C07276=1075.846,98.114,431.514,173.695,23.921,154.199
C07277=1075.840,97.865,431.531,173.693,23.918,154.199
C07278=1075.835,97.616,431.551,173.692,23.916,154.199
C07279=1075.829,97.367,431.568,173.691,23.913,154.198
C07280=1075.823,97.118,431.587,173.688,23.910,154.198
C07281=1075.817,96.868,431.605,173.687,23.908,154.198
C07282=1075.812,96.619,431.624,173.686,23.906,154.198
C07283=1075.805,96.370,431.642,173.683,23.903,154.197
C07284=1075.800,96.121,431.660,173.682,23.901,154.197
C07285=1075.794,95.871,431.678,173.681,23.898,154.197
C07286=1075.789,95.622,431.697,173.679,23.896,154.196
C07287=1075.782,95.341,431.718,173.677,23.893,154.196
C07288=1075.775,95.059,431.738,173.675,23.890,154.196
C07289=1075.770,94.778,431.759,173.674,23.887,154.196
C07290=1075.763,94.497,431.780,173.672,23.884,154.195
C07291=1075.757,94.248,431.797,173.670,23.882,154.195
C07292=1075.751,93.998,431.815,173.669,23.879,154.195
C07293=1075.746,93.749,431.835,173.667,23.877,154.194
C07294=1075.740,93.500,431.852,173.665,23.874,154.194
C07295=1075.734,93.250,431.870,173.664,23.872,154.194
C07296=1075.729,93.001,431.889,173.662,23.869,154.193
C07297=1075.723,92.752,431.907,173.661,23.866,154.193
C07298=1075.717,92.503,431.924,173.659,23.864,154.193
C07299=1075.711,92.253,431.944,173.657,23.861,154.192
C07300=1075.706,92.004,431.961,173.656,23.859,154.192
C07301=1075.700,91.754,431.979,173.655,23.856,154.192
C07302=1075.695,91.506,431.998,173.653,23.854,154.192
C07303=1075.689,91.257,432.016,173.651,23.851,154.191
C07304=1075.683,91.007,432.034,173.650,23.848,154.191
C07305=1075.677,90.758,432.052,173.648,23.846,154.191
C07306=1075.672,90.508,432.070,173.646,23.843,154.190
C07307=1075.666,90.259,432.088,173.645,23.841,154.190
C07308=1075.660,90.010,432.106,173.644,23.838,154.190
C07309=1075.654,89.760,432.124,173.642,23.836,154.190
C07310=1075.648,89.511,432.142,173.640,23.833,154.189
C07311=1075.642,89.262,432.160,173.639,23.831,154.189
C07312=1075.637,89.013,432.178,173.637,23.829,154.189
C07313=1075.630,88.764,432.196,173.635,23.826,154.188
C07314=1075.625,88.514,432.214,173.634,23.823,154.188
C07315=1075.619,88.264,432.232,173.632,23.821,154.188
C07316=1075.614,88.015,432.250,173.630,23.818,154.188
C07317=1075.608,87.766,432.267,173.629,23.816,154.187
C07318=1075.602,87.517,432.285,173.628,23.814,154.187
C07319=1075.596,87.268,432.304,173.626,23.811,154.187
C07320=1075.590,87.018,432.322,173.624,23.808,154.186
C07321=1075.585,86.769,432.339,173.623,23.806,154.186
C07322=1075.579,86.520,432.357,173.622,23.803,154.186
C07323=1075.573,86.271,432.375,173.620,23.801,154.185
C07324=1075.567,86.021,432.393,173.618,23.798,154.185
C07325=1075.561,85.772,432.410,173.617,23.796,154.185
C07326=1075.555,85.523,432.429,173.615,23.793,154.185
C07327=1075.549,85.274,432.446,173.613,23.791,154.184
C07328=1075.544,85.025,432.464,173.612,23.788,154.184
C07329=1075.538,84.775,432.482,173.611,23.785,154.184
C07330=1075.532,84.526,432.499,173.609,23.783,154.183
C07331=1075.527,84.276,432.518,173.607,23.780,154.183
C07332=1075.521,84.027,432.536,173.606,23.778,154.183
C07333=1075.516,83.778,432.553,173.604,23.775,154.183
C07334=1075.510,83.528,432.571,173.603,23.773,154.182
C07335=1075.504,83.279,432.589,173.601,23.770,154.182
C07336=1075.498,83.029,432.607,173.600,23.767,154.182
C07337=1075.493,82.780,432.624,173.598,23.765,154.181
C07338=1075.487,82.531,432.642,173.596,23.762,154.181
C07339=1075.481,82.281,432.660,173.595,23.760,154.181
C07340=1075.475,82.032,432.677,173.593,23.757,154.180
C07341=1075.470,81.783,432.695,173.592,23.755,154.180
C07342=1075.464,81.534,432.713,173.590,23.752,154.180
C07343=1075.458,81.285,432.730,173.589,23.749,154.180
C07344=1075.453,81.035,432.748,173.587,23.747,154.179
C07345=1075.447,80.786,432.766,173.586,23.745,154.179
C07346=1075.441,80.537,432.783,173.584,23.742,154.179
C07347=1075.436,80.288,432.801,173.583,23.739,154.178
C07348=1075.430,80.038,432.819,173.581,23.736,154.178
C07349=1075.424,79.789,432.836,173.580,23.734,154.178
C07350=1075.419,79.539,432.853,173.578,23.731,154.177
C07351=1075.412,79.258,432.874,173.577,23.728,154.177
C07352=1075.405,78.977,432.893,173.574,23.726,154.177
C07353=1075.399,78.696,432.912,173.573,23.723,154.176
C07354=1075.392,78.414,432.933,173.571,23.720,154.176
C07355=1075.387,78.165,432.950,173.570,23.718,154.176
C07356=1075.381,77.916,432.968,173.569,23.715,154.175
C07357=1075.375,77.666,432.986,173.566,23.712,154.175
C07358=1075.369,77.417,433.002,173.565,23.710,154.175
C07359=1075.364,77.168,433.020,173.564,23.707,154.175
C07360=1075.358,76.918,433.038,173.562,23.705,154.174
C07361=1075.352,76.669,433.055,173.560,23.702,154.174
C07362=1075.346,76.420,433.073,173.559,23.700,154.174
C07363=1075.340,76.170,433.089,173.558,23.697,154.173
C07364=1075.334,75.921,433.107,173.556,23.694,154.173
C07365=1075.329,75.672,433.124,173.554,23.692,154.173
C07366=1075.323,75.422,433.142,173.553,23.689,154.172
C07367=1075.317,75.173,433.159,173.552,23.687,154.172
C07368=1075.311,74.924,433.176,173.550,23.684,154.172
C07369=1075.306,74.675,433.194,173.548,23.682,154.172
C07370=1075.300,74.425,433.212,173.547,23.679,154.171
C07371=1075.294,74.176,433.228,173.546,23.676,154.171
C07372=1075.288,73.926,433.246,173.544,23.674,154.171
C07373=1075.282,73.677,433.263,173.542,23.671,154.170
C07374=1075.277,73.427,433.280,173.541,23.669,154.170
C07375=1075.271,73.178,433.297,173.539,23.666,154.170
C07376=1075.265,72.929,433.315,173.538,23.664,154.170
C07377=1075.259,72.680,433.333,173.536,23.661,154.169
C07378=1075.254,72.430,433.350,173.535,23.658,154.169
C07379=1075.247,72.181,433.367,173.533,23.656,154.169
C07380=1075.242,71.932,433.383,173.532,23.653,154.168
C07381=1075.236,71.682,433.401,173.531,23.651,154.168
C07382=1075.230,71.433,433.418,173.529,23.648,154.168
C07383=1075.225,71.183,433.435,173.527,23.645,154.167
C07384=1075.219,70.934,433.453,173.526,23.643,154.167
C07385=1075.214,70.685,433.470,173.525,23.641,154.167
C07386=1075.207,70.435,433.487,173.523,23.638,154.166
C07387=1075.202,70.186,433.505,173.521,23.635,154.166
C07388=1075.196,69.937,433.521,173.520,23.633,154.166
C07389=1075.190,69.688,433.538,173.519,23.630,154.165
C07390=1075.184,69.437,433.556,173.517,23.627,154.165
C07391=1075.178,69.189,433.573,173.515,23.625,154.165
C07392=1075.173,68.940,433.590,173.514,23.623,154.165
C07393=1075.167,68.690,433.607,173.513,23.620,154.164
C07394=1075.161,68.441,433.624,173.511,23.617,154.164
C07395=1075.155,68.191,433.641,173.509,23.615,154.164
C07396=1075.149,67.942,433.658,173.508,23.612,154.163
C07397=1075.144,67.693,433.675,173.507,23.610,154.163
C07398=1075.138,67.444,433.693,173.505,23.607,154.163
C07399=1075.132,67.194,433.709,173.503,23.605,154.163
C07400=1075.126,66.944,433.727,173.502,23.602,154.162
C07401=1075.120,66.695,433.743,173.501,23.599,154.162
C07402=1075.115,66.446,433.761,173.499,23.597,154.162
C07403=1075.109,66.197,433.777,173.497,23.594,154.161
C07404=1075.104,65.947,433.794,173.496,23.592,154.161
C07405=1075.097,65.698,433.811,173.495,23.589,154.161
C07406=1075.091,65.448,433.828,173.493,23.586,154.160
C07407=1075.085,65.199,433.845,173.492,23.584,154.160
C07408=1075.080,64.950,433.862,173.490,23.581,154.160
C07409=1075.074,64.701,433.879,173.489,23.579,154.160
C07410=1075.069,64.451,433.896,173.487,23.576,154.159
C07411=1075.063,64.202,433.912,173.486,23.573,154.159
C07412=1075.056,63.952,433.930,173.485,23.571,154.159
C07413=1075.050,63.703,433.946,173.483,23.568,154.158
C07414=1075.044,63.454,433.963,173.481,23.566,154.158
C07415=1075.038,63.173,433.982,173.480,23.564,154.158
C07416=1075.031,62.892,434.000,173.478,23.560,154.157
C07417=1075.024,62.609,434.020,173.477,23.558,154.157
C07418=1075.018,62.328,434.039,173.475,23.555,154.157
C07419=1075.012,62.079,434.055,173.473,23.552,154.156
C07420=1075.006,61.830,434.071,173.472,23.550,154.156
C07421=1075.000,61.580,434.089,173.470,23.547,154.156
C07422=1074.994,61.330,434.106,173.468,23.545,154.156
C07423=1074.988,61.081,434.122,173.467,23.542,154.155
C07424=1074.983,60.831,434.139,173.466,23.540,154.155
C07425=1074.976,60.583,434.156,173.465,23.537,154.155
C07426=1074.970,60.333,434.172,173.462,23.534,154.154
C07427=1074.964,60.084,434.188,173.461,23.532,154.154
C07428=1074.959,59.834,434.205,173.460,23.529,154.154
C07429=1074.952,59.585,434.222,173.459,23.527,154.153
C07430=1074.946,59.336,434.239,173.457,23.524,154.153
C07431=1074.941,59.086,434.255,173.455,23.522,154.153
C07432=1074.935,58.837,434.272,173.454,23.519,154.153
C07433=1074.929,58.588,434.289,173.453,23.516,154.152
C07434=1074.923,58.338,434.305,173.451,23.514,154.152
C07435=1074.918,58.089,434.322,173.450,23.512,154.152
C07436=1074.912,57.839,434.338,173.448,23.509,154.151
C07437=1074.906,57.590,434.354,173.446,23.506,154.151
C07438=1074.900,57.341,434.371,173.445,23.504,154.151
C07439=1074.894,57.091,434.388,173.444,23.502,154.150
C07440=1074.888,56.842,434.405,173.443,23.499,154.150
C07441=1074.882,56.592,434.421,173.440,23.496,154.150
C07442=1074.876,56.343,434.437,173.439,23.493,154.150
C07443=1074.871,56.093,434.454,173.438,23.491,154.149
C07444=1074.865,55.844,434.470,173.437,23.489,154.149
C07445=1074.859,55.595,434.487,173.435,23.486,154.149
C07446=1074.853,55.345,434.503,173.433,23.483,154.148
C07447=1074.847,55.097,434.520,173.432,23.481,154.148
C07448=1074.841,54.847,434.537,173.431,23.478,154.148
C07449=1074.836,54.598,434.553,173.429,23.476,154.147
C07450=1074.830,54.348,434.569,173.428,23.473,154.147
C07451=1074.824,54.099,434.585,173.426,23.470,154.147
C07452=1074.818,53.849,434.602,173.425,23.468,154.146
C07453=1074.812,53.600,434.619,173.423,23.465,154.146
C07454=1074.807,53.350,434.635,173.422,23.463,154.146
C07455=1074.801,53.101,434.651,173.421,23.460,154.146
C07456=1074.795,52.852,434.667,173.419,23.457,154.145
C07457=1074.789,52.602,434.684,173.417,23.455,154.145
C07458=1074.783,52.353,434.700,173.416,23.452,154.145
C07459=1074.777,52.103,434.717,173.415,23.450,154.144
C07460=1074.772,51.854,434.733,173.414,23.447,154.144
C07461=1074.766,51.605,434.749,173.412,23.444,154.144
C07462=1074.760,51.355,434.765,173.410,23.442,154.143
C07463=1074.754,51.106,434.782,173.409,23.439,154.143
C07464=1074.748,50.856,434.799,173.408,23.437,154.143
C07465=1074.743,50.607,434.815,173.406,23.434,154.142
C07466=1074.737,50.358,434.831,173.404,23.431,154.142
C07467=1074.731,50.108,434.847,173.403,23.429,154.142
C07468=1074.725,49.859,434.864,173.402,23.426,154.142
C07469=1074.719,49.609,434.880,173.400,23.424,154.141
C07470=1074.714,49.360,434.897,173.399,23.421,154.141
C07471=1074.708,49.111,434.912,173.398,23.419,154.141
C07472=1074.703,48.861,434.928,173.396,23.416,154.140
C07473=1074.697,48.612,434.944,173.394,23.413,154.140
C07474=1074.691,48.363,434.961,173.393,23.411,154.140
C07475=1074.685,48.113,434.977,173.392,23.408,154.139
C07476=1074.679,47.864,434.994,173.391,23.406,154.139
C07477=1074.673,47.614,435.010,173.389,23.403,154.139
C07478=1074.668,47.365,435.026,173.387,23.400,154.138
C07479=1074.661,47.083,435.044,173.386,23.398,154.138
C07480=1074.655,46.801,435.062,173.384,23.394,154.138
C07481=1074.648,46.520,435.081,173.383,23.391,154.137
C07482=1074.642,46.238,435.099,173.381,23.389,154.137
C07483=1074.636,45.989,435.115,173.380,23.386,154.137
C07484=1074.630,45.739,435.131,173.378,23.383,154.136
C07485=1074.625,45.490,435.147,173.377,23.381,154.136
C07486=1074.619,45.241,435.163,173.376,23.378,154.136
C07487=1074.614,44.991,435.180,173.374,23.375,154.135
C07488=1074.608,44.742,435.196,173.372,23.373,154.135
C07489=1074.602,44.492,435.212,173.371,23.370,154.135
C07490=1074.596,44.243,435.228,173.370,23.367,154.134
C07491=1074.591,43.994,435.244,173.369,23.365,154.134
C07492=1074.585,43.744,435.259,173.367,23.362,154.134
C07493=1074.579,43.495,435.276,173.365,23.360,154.134
C07494=1074.573,43.245,435.292,173.364,23.357,154.133
C07495=1074.567,42.996,435.308,173.363,23.354,154.133
C07496=1074.562,42.746,435.324,173.362,23.352,154.133
C07497=1074.556,42.497,435.340,173.360,23.349,154.132
C07498=1074.549,42.248,435.356,173.359,23.347,154.132
C07499=1074.544,41.998,435.371,173.357,23.344,154.132
C07500=1074.538,41.749,435.387,173.356,23.341,154.131
C07501=1074.532,41.500,435.403,173.354,23.339,154.131
C07502=1074.526,41.250,435.419,173.353,23.337,154.131
C07503=1074.520,41.000,435.435,173.352,23.334,154.131
C07504=1074.515,40.751,435.451,173.350,23.332,154.130
C07505=1074.509,40.501,435.467,173.348,23.328,154.130
C07506=1074.504,40.252,435.483,173.347,23.326,154.130
C07507=1074.497,40.003,435.498,173.346,23.324,154.129
C07508=1074.491,39.753,435.514,173.345,23.321,154.129
C07509=1074.485,39.504,435.530,173.343,23.318,154.129
C07510=1074.480,39.254,435.546,173.341,23.315,154.128
C07511=1074.474,39.005,435.562,173.340,23.313,154.128
C07512=1074.469,38.755,435.577,173.339,23.311,154.128
C07513=1074.463,38.506,435.593,173.337,23.308,154.127
C07514=1074.457,38.256,435.609,173.336,23.305,154.127
C07515=1074.450,38.007,435.625,173.335,23.303,154.127
C07516=1074.445,37.758,435.640,173.333,23.300,154.127
C07517=1074.439,37.508,435.656,173.332,23.298,154.126
C07518=1074.433,37.259,435.672,173.330,23.295,154.126
C07519=1074.427,37.009,435.687,173.329,23.293,154.126
C07520=1074.421,36.760,435.703,173.328,23.290,154.125
C07521=1074.415,36.510,435.719,173.327,23.287,154.125
C07522=1074.409,36.262,435.734,173.324,23.285,154.125
C07523=1074.404,36.012,435.750,173.323,23.282,154.124
C07524=1074.398,35.762,435.766,173.322,23.280,154.124
C07525=1074.392,35.513,435.782,173.320,23.277,154.124
C07526=1074.386,35.263,435.797,173.319,23.275,154.124
C07527=1074.380,35.014,435.812,173.318,23.272,154.123
C07528=1074.375,34.764,435.828,173.316,23.269,154.123
C07529=1074.368,34.515,435.844,173.315,23.267,154.123
C07530=1074.362,34.265,435.859,173.313,23.264,154.122
C07531=1074.357,34.017,435.875,173.312,23.262,154.122
C07532=1074.351,33.767,435.890,173.311,23.260,154.122
C07533=1074.345,33.517,435.906,173.309,23.257,154.121
C07534=1074.339,33.268,435.922,173.308,23.254,154.121
C07535=1074.333,33.019,435.936,173.306,23.251,154.121
C07536=1074.327,32.769,435.953,173.305,23.249,154.120
C07537=1074.322,32.519,435.968,173.304,23.247,154.120
C07538=1074.315,32.270,435.983,173.302,23.244,154.120
C07539=1074.310,32.021,435.999,173.301,23.242,154.120
C07540=1074.304,31.771,436.015,173.300,23.239,154.119
C07541=1074.298,31.521,436.030,173.298,23.236,154.119
C07542=1074.292,31.272,436.046,173.296,23.234,154.119
C07543=1074.285,30.991,436.063,173.295,23.231,154.118
C07544=1074.279,30.709,436.080,173.293,23.228,154.118
C07545=1074.272,30.427,436.098,173.292,23.225,154.118
C07546=1074.265,30.146,436.115,173.291,23.222,154.117
C07547=1074.260,29.897,436.130,173.289,23.220,154.117
C07548=1074.255,29.647,436.146,173.287,23.217,154.117
C07549=1074.248,29.398,436.161,173.286,23.214,154.116
C07550=1074.243,29.148,436.177,173.285,23.212,154.116
C07551=1074.237,28.898,436.192,173.284,23.209,154.116
C07552=1074.230,28.649,436.208,173.282,23.207,154.116
C07553=1074.225,28.400,436.223,173.280,23.204,154.115
C07554=1074.219,28.150,436.238,173.279,23.201,154.115
C07555=1074.213,27.900,436.253,173.278,23.199,154.115
C07556=1074.207,27.651,436.268,173.276,23.196,154.114
C07557=1074.202,27.402,436.284,173.275,23.194,154.114
C07558=1074.195,27.152,436.299,173.274,23.192,154.114
C07559=1074.190,26.902,436.315,173.273,23.189,154.113
C07560=1074.184,26.653,436.329,173.270,23.186,154.113
C07561=1074.178,26.404,436.345,173.269,23.184,154.113
C07562=1074.172,26.154,436.360,173.268,23.181,154.112
C07563=1074.166,25.906,436.375,173.267,23.178,154.112
C07564=1074.160,25.656,436.391,173.265,23.176,154.112
C07565=1074.154,25.406,436.406,173.264,23.174,154.112
C07566=1074.149,25.157,436.421,173.263,23.171,154.111
C07567=1074.142,24.907,436.436,173.261,23.168,154.111
C07568=1074.137,24.657,436.451,173.259,23.166,154.111
C07569=1074.131,24.409,436.467,173.258,23.164,154.111
C07570=1074.124,24.159,436.481,173.257,23.161,154.110
C07571=1074.119,23.909,436.497,173.256,23.158,154.110
C07572=1074.113,23.660,436.512,173.255,23.156,154.110
C07573=1074.107,23.410,436.527,173.252,23.153,154.109
C07574=1074.101,23.160,436.542,173.251,23.151,154.109
C07575=1074.095,22.912,436.557,173.250,23.148,154.109
C07576=1074.089,22.662,436.572,173.248,23.146,154.108
C07577=1074.083,22.413,436.587,173.247,23.143,154.108
C07578=1074.078,22.163,436.602,173.246,23.141,154.108
C07579=1074.071,21.913,436.617,173.245,23.138,154.107
C07580=1074.066,21.664,436.632,173.243,23.135,154.107
C07581=1074.060,21.414,436.647,173.241,23.133,154.107
C07582=1074.054,21.165,436.662,173.240,23.130,154.107
C07583=1074.049,20.915,436.678,173.239,23.128,154.106
C07584=1074.042,20.665,436.692,173.238,23.125,154.106
C07585=1074.036,20.417,436.707,173.236,23.123,154.106
C07586=1074.031,20.167,436.723,173.235,23.121,154.105
C07587=1074.025,19.918,436.737,173.233,23.118,154.105
C07588=1074.019,19.668,436.752,173.232,23.115,154.105
C07589=1074.013,19.418,436.768,173.230,23.112,154.105
C07590=1074.007,19.169,436.782,173.229,23.110,154.104
C07591=1074.001,18.919,436.797,173.228,23.108,154.104
C07592=1073.995,18.670,436.812,173.227,23.105,154.104
C07593=1073.989,18.420,436.827,173.225,23.103,154.103
C07594=1073.984,18.171,436.842,173.223,23.100,154.103
C07595=1073.977,17.922,436.857,173.222,23.097,154.103
C07596=1073.971,17.672,436.872,173.221,23.095,154.103
C07597=1073.966,17.423,436.887,173.219,23.093,154.102
C07598=1073.960,17.173,436.901,173.218,23.090,154.102
C07599=1073.954,16.924,436.916,173.217,23.088,154.102
C07600=1073.948,16.674,436.931,173.216,23.085,154.101
C07601=1073.943,16.425,436.946,173.214,23.082,154.101
C07602=1073.936,16.175,436.961,173.212,23.080,154.101
C07603=1073.930,15.926,436.975,173.211,23.077,154.100
C07604=1073.924,15.676,436.990,173.210,23.075,154.100
C07605=1073.919,15.427,437.006,173.208,23.072,154.100
C07606=1073.913,15.177,437.020,173.207,23.070,154.100
C07607=1073.906,14.897,437.036,173.205,23.066,154.099
C07608=1073.900,14.616,437.053,173.204,23.064,154.099
C07609=1073.893,14.337,437.069,173.203,23.062,154.099
C07610=1073.886,14.056,437.087,173.201,23.058,154.098
C07611=1073.881,13.807,437.101,173.199,23.056,154.098
C07612=1073.874,13.557,437.116,173.198,23.053,154.098
C07613=1073.868,13.308,437.130,173.197,23.051,154.097
C07614=1073.862,13.059,437.145,173.196,23.049,154.097
C07615=1073.856,12.808,437.159,173.194,23.046,154.097
C07616=1073.850,12.559,437.174,173.192,23.043,154.097
C07617=1073.844,12.310,437.189,173.191,23.041,154.096
C07618=1073.838,12.061,437.203,173.190,23.038,154.096
C07619=1073.832,11.810,437.218,173.188,23.036,154.096
C07620=1073.826,11.561,437.232,173.187,23.034,154.095
C07621=1073.820,11.312,437.247,173.186,23.031,154.095
C07622=1073.815,11.062,437.261,173.184,23.029,154.095
C07623=1073.808,10.813,437.276,173.182,23.026,154.095
C07624=1073.802,10.564,437.291,173.181,23.024,154.094
C07625=1073.796,10.313,437.305,173.180,23.021,154.094
C07626=1073.790,10.064,437.319,173.179,23.019,154.094
C07627=1073.784,9.815,437.334,173.177,23.016,154.094
C07628=1073.779,9.565,437.348,173.176,23.014,154.093
C07629=1073.772,9.316,437.363,173.175,23.011,154.093
C07630=1073.766,9.067,437.378,173.173,23.009,154.093
C07631=1073.760,8.816,437.392,173.171,23.006,154.092
C07632=1073.755,8.567,437.407,173.170,23.004,154.092
C07633=1073.748,8.318,437.421,173.169,23.002,154.092
C07634=1073.743,8.068,437.435,173.167,22.999,154.092
C07635=1073.736,7.818,437.450,173.166,22.997,154.091
C07636=1073.731,7.569,437.464,173.165,22.995,154.091
C07637=1073.725,7.320,437.479,173.163,22.992,154.091
C07638=1073.719,7.070,437.494,173.161,22.989,154.091
C07639=1073.713,6.821,437.508,173.160,22.987,154.090
C07640=1073.707,6.571,437.522,173.159,22.984,154.090
C07641=1073.701,6.321,437.536,173.158,22.982,154.090
C07642=1073.695,6.072,437.551,173.156,22.980,154.089
C07643=1073.690,5.822,437.565,173.155,22.977,154.089
C07644=1073.684,5.573,437.580,173.154,22.975,154.089
C07645=1073.678,5.323,437.594,173.152,22.972,154.089
C07646=1073.672,5.074,437.609,173.150,22.969,154.088
C07647=1073.666,4.824,437.623,173.149,22.967,154.088
C07648=1073.659,4.575,437.637,173.148,22.965,154.088
C07649=1073.654,4.326,437.651,173.146,22.962,154.087
C07650=1073.647,4.076,437.666,173.145,22.960,154.087
C07651=1073.642,3.826,437.679,173.144,22.957,154.087
C07652=1073.636,3.577,437.694,173.143,22.955,154.087
C07653=1073.630,3.327,437.708,173.141,22.952,154.086
C07654=1073.624,3.078,437.723,173.139,22.950,154.086
C07655=1073.618,2.828,437.737,173.138,22.947,154.086
C07656=1073.612,2.579,437.752,173.137,22.945,154.086
C07657=1073.607,2.329,437.765,173.135,22.942,154.085
C07658=1073.601,2.079,437.780,173.134,22.940,154.085
C07659=1073.595,1.830,437.794,173.133,22.937,154.085
C07660=1073.590,1.581,437.808,173.132,22.935,154.084
C07661=1073.583,1.331,437.823,173.130,22.933,154.084
C07662=1073.577,1.082,437.836,173.128,22.930,154.084
C07663=1073.572,0.832,437.850,173.127,22.927,154.084
C07664=1073.565,0.582,437.865,173.126,22.925,154.083
C07665=1073.560,0.333,437.879,173.124,22.922,154.083
C07666=1073.554,0.084,437.894,173.123,22.920,154.083
C07667=1073.548,-0.166,437.908,173.122,22.918,154.082
C07668=1073.542,-0.416,437.922,173.121,22.915,154.082
C07669=1073.537,-0.665,437.936,173.119,22.913,154.082
C07670=1073.531,-0.915,437.950,173.117,22.910,154.082
C07671=1073.524,-1.193,437.966,173.116,22.907,154.081
C07672=1073.517,-1.471,437.981,173.115,22.904,154.081
C07673=1073.511,-1.750,437.998,173.113,22.902,154.081
C07674=1073.504,-2.027,438.013,173.112,22.899,154.080
C07675=1073.498,-2.278,438.027,173.110,22.897,154.080
C07676=1073.493,-2.527,438.041,173.109,22.894,154.080
C07677=1073.487,-2.777,438.055,173.108,22.892,154.080
C07678=1073.482,-3.026,438.070,173.106,22.889,154.079
C07679=1073.476,-3.276,438.084,173.104,22.887,154.079
C07680=1073.469,-3.525,438.097,173.103,22.884,154.079
C07681=1073.464,-3.775,438.111,173.102,22.882,154.078
C07682=1073.457,-4.024,438.125,173.101,22.879,154.078
C07683=1073.451,-4.274,438.139,173.099,22.877,154.078
C07684=1073.446,-4.523,438.153,173.098,22.874,154.078
C07685=1073.439,-4.773,438.167,173.097,22.873,154.077
C07686=1073.433,-5.022,438.181,173.094,22.870,154.077
C07687=1073.428,-5.272,438.195,173.093,22.867,154.077
C07688=1073.422,-5.521,438.208,173.092,22.865,154.077
C07689=1073.415,-5.771,438.223,173.091,22.862,154.076
C07690=1073.409,-6.021,438.236,173.089,22.860,154.076
C07691=1073.404,-6.270,438.250,173.088,22.858,154.076
C07692=1073.397,-6.520,438.265,173.087,22.856,154.076
C07693=1073.391,-6.769,438.278,173.085,22.853,154.075
C07694=1073.386,-7.019,438.292,173.083,22.850,154.075
C07695=1073.379,-7.268,438.305,173.082,22.848,154.075
C07696=1073.373,-7.518,438.319,173.081,22.845,154.075
C07697=1073.368,-7.768,438.333,173.080,22.843,154.074
C07698=1073.362,-8.017,438.346,173.078,22.841,154.074
C07699=1073.356,-8.266,438.361,173.077,22.839,154.074
C07700=1073.349,-8.516,438.375,173.076,22.836,154.074
C07701=1073.344,-8.765,438.389,173.074,22.834,154.073
C07702=1073.338,-9.015,438.402,173.073,22.831,154.073
C07703=1073.332,-9.264,438.416,173.071,22.829,154.073
C07704=1073.326,-9.515,438.430,173.069,22.827,154.073
C07705=1073.320,-9.764,438.443,173.068,22.824,154.072
C07706=1073.314,-10.013,438.457,173.067,22.822,154.072
C07707=1073.308,-10.263,438.470,173.066,22.819,154.072
C07708=1073.302,-10.512,438.484,173.064,22.817,154.071
C07709=1073.296,-10.763,438.498,173.063,22.815,154.071
C07710=1073.290,-11.012,438.512,173.062,22.813,154.071
C07711=1073.285,-11.261,438.526,173.060,22.810,154.071
C07712=1073.278,-11.511,438.539,173.058,22.807,154.070
C07713=1073.273,-11.760,438.553,173.057,22.805,154.070
C07714=1073.266,-12.010,438.566,173.056,22.802,154.070
C07715=1073.261,-12.260,438.580,173.054,22.801,154.070
C07716=1073.254,-12.509,438.593,173.053,22.798,154.069
C07717=1073.249,-12.759,438.607,173.052,22.796,154.069
C07718=1073.243,-13.008,438.621,173.051,22.793,154.069
C07719=1073.237,-13.257,438.634,173.049,22.791,154.069
C07720=1073.231,-13.507,438.648,173.047,22.788,154.069
C07721=1073.225,-13.757,438.662,173.046,22.786,154.068
C07722=1073.220,-14.007,438.676,173.045,22.784,154.068
C07723=1073.213,-14.256,438.689,173.043,22.781,154.068
C07724=1073.208,-14.505,438.703,173.042,22.779,154.067
C07725=1073.202,-14.755,438.716,173.041,22.777,154.067
C07726=1073.196,-15.004,438.730,173.039,22.774,154.067
C07727=1073.190,-15.254,438.743,173.038,22.772,154.067
C07728=1073.183,-15.504,438.756,173.036,22.769,154.066
C07729=1073.178,-15.754,438.770,173.035,22.767,154.066
C07730=1073.172,-16.003,438.783,173.033,22.765,154.066
C07731=1073.166,-16.252,438.797,173.032,22.762,154.066
C07732=1073.160,-16.502,438.811,173.031,22.760,154.066
C07733=1073.154,-16.751,438.824,173.029,22.758,154.065
C07734=1073.147,-17.002,438.837,173.028,22.756,154.065
C07735=1073.141,-17.278,438.853,173.026,22.753,154.065
C07736=1073.135,-17.554,438.867,173.025,22.750,154.064
C07737=1073.127,-17.831,438.882,173.023,22.748,154.064
C07738=1073.121,-18.108,438.896,173.021,22.745,154.064
C07739=1073.115,-18.357,438.910,173.020,22.743,154.064
C07740=1073.109,-18.607,438.923,173.019,22.741,154.063
C07741=1073.103,-18.856,438.936,173.017,22.738,154.063
C07742=1073.098,-19.106,438.950,173.016,22.736,154.063
C07743=1073.091,-19.355,438.963,173.015,22.734,154.063
C07744=1073.085,-19.605,438.977,173.013,22.731,154.062
C07745=1073.079,-19.855,438.989,173.012,22.729,154.062
C07746=1073.073,-20.105,439.003,173.011,22.727,154.062
C07747=1073.067,-20.354,439.017,173.009,22.724,154.062
C07748=1073.061,-20.604,439.029,173.007,22.722,154.062
C07749=1073.056,-20.853,439.043,173.006,22.720,154.061
C07750=1073.049,-21.103,439.056,173.005,22.717,154.061
C07751=1073.043,-21.352,439.070,173.004,22.715,154.061
C07752=1073.037,-21.602,439.082,173.002,22.713,154.061
C07753=1073.032,-21.851,439.096,173.001,22.711,154.060
C07754=1073.026,-22.100,439.109,173.000,22.708,154.060
C07755=1073.020,-22.350,439.122,172.998,22.706,154.060
C07756=1073.013,-22.600,439.135,172.996,22.703,154.060
C07757=1073.008,-22.849,439.149,172.995,22.701,154.059
C07758=1073.001,-23.100,439.162,172.993,22.699,154.059
C07759=1072.995,-23.349,439.175,172.992,22.697,154.059
C07760=1072.990,-23.599,439.189,172.991,22.694,154.059
C07761=1072.984,-23.849,439.202,172.989,22.692,154.059
C07762=1072.978,-24.098,439.215,172.988,22.690,154.058
C07763=1072.971,-24.347,439.228,172.987,22.688,154.058
C07764=1072.966,-24.597,439.241,172.985,22.685,154.058
C07765=1072.960,-24.847,439.254,172.983,22.683,154.058
C07766=1072.954,-25.096,439.267,172.982,22.681,154.057
C07767=1072.948,-25.346,439.280,172.981,22.678,154.057
C07768=1072.942,-25.595,439.294,172.979,22.676,154.057
C07769=1072.937,-25.845,439.307,172.978,22.674,154.057
C07770=1072.930,-26.094,439.320,172.977,22.671,154.056
C07771=1072.924,-26.344,439.333,172.976,22.669,154.056
C07772=1072.918,-26.594,439.346,172.974,22.667,154.056
C07773=1072.913,-26.844,439.359,172.973,22.665,154.056
C07774=1072.907,-27.093,439.372,172.971,22.662,154.056
C07775=1072.901,-27.343,439.385,172.969,22.660,154.055
C07776=1072.895,-27.592,439.398,172.968,22.658,154.055
C07777=1072.889,-27.842,439.411,172.967,22.656,154.055
C07778=1072.883,-28.091,439.424,172.965,22.654,154.055
C07779=1072.877,-28.341,439.436,172.964,22.651,154.054
C07780=1072.870,-28.590,439.450,172.963,22.649,154.054
C07781=1072.865,-28.840,439.462,172.961,22.647,154.054
C07782=1072.858,-29.090,439.476,172.960,22.645,154.054
C07783=1072.852,-29.339,439.488,172.959,22.643,154.054
C07784=1072.846,-29.589,439.501,172.956,22.640,154.053
C07785=1072.840,-29.839,439.514,172.955,22.638,154.053
C07786=1072.834,-30.088,439.527,172.954,22.635,154.053
C07787=1072.828,-30.338,439.540,172.952,22.633,154.053
C07788=1072.822,-30.587,439.553,172.951,22.632,154.053
C07789=1072.816,-30.837,439.566,172.950,22.629,154.052
C07790=1072.810,-31.087,439.578,172.948,22.627,154.052
C07791=1072.804,-31.336,439.591,172.947,22.625,154.052
C07792=1072.799,-31.585,439.604,172.946,22.623,154.052
C07793=1072.792,-31.834,439.617,172.944,22.620,154.051
C07794=1072.787,-32.084,439.629,172.942,22.618,154.051
C07795=1072.781,-32.334,439.642,172.941,22.616,154.051
C07796=1072.774,-32.584,439.655,172.939,22.614,154.051
C07797=1072.768,-32.833,439.668,172.938,22.611,154.051
C07798=1072.762,-33.083,439.681,172.937,22.609,154.050
C07799=1072.756,-33.359,439.696,172.936,22.607,154.050
C07800=1072.749,-33.634,439.709,172.933,22.604,154.050
C07801=1072.743,-33.910,439.723,172.932,22.602,154.050
C07802=1072.736,-34.186,439.737,172.931,22.600,154.049
C07803=1072.730,-34.436,439.750,172.929,22.597,154.049
C07804=1072.724,-34.686,439.762,172.928,22.595,154.049
C07805=1072.717,-34.935,439.776,172.926,22.592,154.049
C07806=1072.712,-35.184,439.788,172.925,22.591,154.049
C07807=1072.706,-35.434,439.800,172.923,22.588,154.048
C07808=1072.700,-35.683,439.814,172.922,22.586,154.048
C07809=1072.694,-35.933,439.826,172.920,22.584,154.048
C07810=1072.688,-36.183,439.839,172.919,22.582,154.048
C07811=1072.682,-36.433,439.851,172.918,22.580,154.048
C07812=1072.676,-36.682,439.864,172.917,22.577,154.047
C07813=1072.670,-36.932,439.877,172.915,22.576,154.047
C07814=1072.665,-37.181,439.889,172.914,22.573,154.047
C07815=1072.659,-37.431,439.902,172.912,22.571,154.047
C07816=1072.653,-37.681,439.914,172.910,22.569,154.047
C07817=1072.647,-37.930,439.928,172.909,22.566,154.046
C07818=1072.640,-38.180,439.940,172.907,22.565,154.046
C07819=1072.634,-38.430,439.952,172.906,22.562,154.046
C07820=1072.629,-38.679,439.964,172.905,22.560,154.046
C07821=1072.623,-38.929,439.977,172.903,22.558,154.046
C07822=1072.617,-39.178,439.990,172.902,22.556,154.045
C07823=1072.610,-39.428,440.002,172.901,22.554,154.045
C07824=1072.604,-39.678,440.015,172.899,22.552,154.045
C07825=1072.598,-39.928,440.027,172.897,22.549,154.045
C07826=1072.593,-40.177,440.040,172.896,22.547,154.045
C07827=1072.586,-40.427,440.052,172.894,22.545,154.045
C07828=1072.580,-40.676,440.065,172.893,22.543,154.044
C07829=1072.574,-40.926,440.077,172.892,22.541,154.044
C07830=1072.568,-41.175,440.090,172.890,22.539,154.044
C07831=1072.562,-41.425,440.102,172.889,22.537,154.044
C07832=1072.556,-41.675,440.114,172.888,22.535,154.043
C07833=1072.550,-41.925,440.127,172.886,22.533,154.043
C07834=1072.545,-42.174,440.139,172.885,22.531,154.043
C07835=1072.538,-42.423,440.151,172.884,22.528,154.043
C07836=1072.532,-42.673,440.163,172.881,22.526,154.043
C07837=1072.526,-42.923,440.176,172.880,22.524,154.043
C07838=1072.520,-43.173,440.188,172.878,22.522,154.043
C07839=1072.514,-43.421,440.201,172.877,22.520,154.042
C07840=1072.508,-43.671,440.213,172.876,22.518,154.042
C07841=1072.502,-43.921,440.226,172.874,22.516,154.042
C07842=1072.495,-44.171,440.238,172.873,22.514,154.042
C07843=1072.490,-44.421,440.251,172.872,22.512,154.041
C07844=1072.484,-44.670,440.263,172.870,22.510,154.041
C07845=1072.478,-44.919,440.275,172.869,22.508,154.041
C07846=1072.472,-45.169,440.287,172.868,22.505,154.041
C07847=1072.466,-45.419,440.300,172.865,22.503,154.041
C07848=1072.459,-45.669,440.312,172.864,22.501,154.041
C07849=1072.454,-45.918,440.324,172.862,22.499,154.040
C07850=1072.448,-46.168,440.336,172.861,22.497,154.040
C07851=1072.441,-46.417,440.348,172.860,22.495,154.040
C07852=1072.435,-46.667,440.361,172.858,22.493,154.040
C07853=1072.430,-46.917,440.372,172.857,22.491,154.040
C07854=1072.424,-47.167,440.384,172.856,22.489,154.040
C07855=1072.418,-47.416,440.397,172.854,22.487,154.039
C07856=1072.413,-47.666,440.409,172.853,22.485,154.039
C07857=1072.406,-47.915,440.421,172.852,22.483,154.039
C07858=1072.400,-48.165,440.434,172.850,22.481,154.039
C07859=1072.394,-48.415,440.446,172.848,22.479,154.039
C07860=1072.388,-48.664,440.458,172.847,22.476,154.038
C07861=1072.382,-48.914,440.470,172.845,22.474,154.038
C07862=1072.376,-49.164,440.483,172.844,22.472,154.038
C07863=1072.370,-49.440,440.496,172.842,22.470,154.038
C07864=1072.363,-49.716,440.509,172.841,22.468,154.038
C07865=1072.357,-49.992,440.523,172.839,22.466,154.038
C07866=1072.350,-50.269,440.536,172.838,22.463,154.037
C07867=1072.344,-50.518,440.548,172.836,22.461,154.037
C07868=1072.338,-50.767,440.560,172.835,22.459,154.037
C07869=1072.331,-51.018,440.572,172.833,22.458,154.037
C07870=1072.325,-51.267,440.584,172.832,22.456,154.037
C07871=1072.319,-51.516,440.596,172.830,22.454,154.037
C07872=1072.313,-51.766,440.608,172.828,22.451,154.037
C07873=1072.307,-52.016,440.620,172.827,22.450,154.036
C07874=1072.300,-52.266,440.632,172.825,22.448,154.036
C07875=1072.294,-52.515,440.643,172.824,22.446,154.036
C07876=1072.289,-52.765,440.656,172.822,22.444,154.036
C07877=1072.282,-53.014,440.668,172.821,22.442,154.036
C07878=1072.275,-53.264,440.680,172.820,22.440,154.036
C07879=1072.270,-53.514,440.691,172.818,22.438,154.035
C07880=1072.264,-53.763,440.703,172.817,22.436,154.035
C07881=1072.258,-54.013,440.716,172.815,22.434,154.035
C07882=1072.252,-54.262,440.727,172.814,22.432,154.035
C07883=1072.245,-54.512,440.738,172.813,22.430,154.035
C07884=1072.239,-54.762,440.751,172.811,22.428,154.035
C07885=1072.233,-55.012,440.763,172.809,22.426,154.035
C07886=1072.227,-55.261,440.774,172.807,22.424,154.034
C07887=1072.221,-55.511,440.786,172.806,22.422,154.034
C07888=1072.214,-55.761,440.798,172.805,22.420,154.034
C07889=1072.209,-56.010,440.809,172.803,22.419,154.034
C07890=1072.203,-56.260,440.822,172.802,22.417,154.034
C07891=1072.196,-56.510,440.834,172.800,22.415,154.034
C07892=1072.190,-56.759,440.845,172.799,22.413,154.034
C07893=1072.184,-57.009,440.857,172.798,22.411,154.033
C07894=1072.178,-57.258,440.869,172.796,22.410,154.033
C07895=1072.172,-57.508,440.880,172.795,22.408,154.033
C07896=1072.165,-57.758,440.892,172.793,22.406,154.033
C07897=1072.160,-58.007,440.905,172.792,22.404,154.033
C07898=1072.154,-58.257,440.915,172.790,22.402,154.033
C07899=1072.147,-58.507,440.927,172.788,22.400,154.033
C07900=1072.142,-58.756,440.939,172.787,22.398,154.033
C07901=1072.136,-59.006,440.951,172.785,22.396,154.032
C07902=1072.129,-59.255,440.963,172.784,22.394,154.032
C07903=1072.123,-59.505,440.974,172.782,22.392,154.032
C07904=1072.117,-59.755,440.986,172.781,22.390,154.032
C07905=1072.111,-60.004,440.997,172.780,22.388,154.032
C07906=1072.105,-60.254,441.009,172.778,22.387,154.032
C07907=1072.099,-60.504,441.021,172.777,22.385,154.032
C07908=1072.093,-60.753,441.032,172.775,22.383,154.031
C07909=1072.087,-61.003,441.044,172.774,22.381,154.031
C07910=1072.081,-61.252,441.055,172.772,22.379,154.031
C07911=1072.075,-61.502,441.068,172.771,22.377,154.031
C07912=1072.069,-61.752,441.079,172.769,22.375,154.031
C07913=1072.062,-62.001,441.091,172.768,22.373,154.031
C07914=1072.056,-62.251,441.102,172.766,22.371,154.031
C07915=1072.051,-62.501,441.114,172.764,22.370,154.031
C07916=1072.045,-62.751,441.125,172.763,22.368,154.030
C07917=1072.038,-63.000,441.137,172.761,22.366,154.030
C07918=1072.032,-63.250,441.148,172.760,22.364,154.030
C07919=1072.027,-63.499,441.160,172.759,22.362,154.030
C07920=1072.020,-63.749,441.172,172.757,22.360,154.030
C07921=1072.014,-63.999,441.183,172.756,22.359,154.030
C07922=1072.008,-64.248,441.195,172.754,22.357,154.030
C07923=1072.002,-64.499,441.206,172.753,22.355,154.029
C07924=1071.996,-64.748,441.218,172.751,22.353,154.029
C07925=1071.990,-64.998,441.229,172.750,22.351,154.029
C07926=1071.984,-65.247,441.241,172.748,22.349,154.029
C07927=1071.978,-65.524,441.254,172.746,22.347,154.029
C07928=1071.971,-65.802,441.267,172.745,22.345,154.029
C07929=1071.964,-66.080,441.279,172.743,22.343,154.029
C07930=1071.957,-66.357,441.292,172.742,22.341,154.028
C07931=1071.952,-66.607,441.303,172.740,22.340,154.028
C07932=1071.946,-66.857,441.314,172.738,22.337,154.028
C07933=1071.940,-67.106,441.326,172.737,22.335,154.028
C07934=1071.933,-67.356,441.337,172.735,22.334,154.028
C07935=1071.928,-67.606,441.348,172.734,22.332,154.028
C07936=1071.922,-67.855,441.361,172.732,22.330,154.028
C07937=1071.916,-68.105,441.372,172.731,22.328,154.028
C07938=1071.910,-68.355,441.383,172.729,22.326,154.028
C07939=1071.904,-68.604,441.394,172.728,22.324,154.027
C07940=1071.897,-68.854,441.406,172.727,22.323,154.027
C07941=1071.892,-69.104,441.416,172.725,22.321,154.027
C07942=1071.886,-69.353,441.429,172.724,22.319,154.027
C07943=1071.880,-69.603,441.440,172.722,22.317,154.027
C07944=1071.874,-69.853,441.451,172.721,22.315,154.027
C07945=1071.868,-70.102,441.463,172.719,22.314,154.027
C07946=1071.862,-70.352,441.474,172.718,22.312,154.027
C07947=1071.856,-70.602,441.485,172.716,22.310,154.027
C07948=1071.851,-70.852,441.496,172.715,22.309,154.026
C07949=1071.844,-71.100,441.508,172.713,22.307,154.026
C07950=1071.838,-71.351,441.519,172.712,22.305,154.026
C07951=1071.832,-71.600,441.530,172.711,22.303,154.026
C07952=1071.826,-71.850,441.541,172.708,22.301,154.026
C07953=1071.820,-72.100,441.552,172.707,22.299,154.026
C07954=1071.815,-72.349,441.564,172.705,22.298,154.026
C07955=1071.809,-72.599,441.576,172.704,22.296,154.026
C07956=1071.803,-72.849,441.587,172.702,22.294,154.026
C07957=1071.797,-73.098,441.597,172.701,22.292,154.025
C07958=1071.791,-73.348,441.609,172.699,22.290,154.025
C07959=1071.785,-73.597,441.620,172.698,22.289,154.025
C07960=1071.778,-73.847,441.631,172.696,22.287,154.025
C07961=1071.773,-74.097,441.642,172.695,22.285,154.025
C07962=1071.767,-74.346,441.653,172.693,22.284,154.025
C07963=1071.761,-74.597,441.664,172.692,22.282,154.025
C07964=1071.755,-74.846,441.675,172.690,22.281,154.025
C07965=1071.749,-75.096,441.687,172.689,22.279,154.025
C07966=1071.743,-75.345,441.698,172.687,22.277,154.025
C07967=1071.737,-75.595,441.709,172.686,22.275,154.024
C07968=1071.730,-75.845,441.720,172.684,22.274,154.024
C07969=1071.725,-76.094,441.731,172.683,22.272,154.024
C07970=1071.718,-76.345,441.742,172.681,22.271,154.024
C07971=1071.713,-76.594,441.753,172.680,22.269,154.024
C07972=1071.707,-76.844,441.764,172.678,22.267,154.024
C07973=1071.700,-77.093,441.775,172.677,22.265,154.024
C07974=1071.694,-77.343,441.786,172.675,22.264,154.024
C07975=1071.688,-77.592,441.797,172.674,22.262,154.024
C07976=1071.682,-77.843,441.808,172.672,22.260,154.024
C07977=1071.676,-78.092,441.819,172.670,22.259,154.024
C07978=1071.670,-78.342,441.830,172.669,22.257,154.024
C07979=1071.664,-78.592,441.841,172.667,22.255,154.024
C07980=1071.658,-78.841,441.852,172.666,22.254,154.024
C07981=1071.652,-79.091,441.864,172.664,22.252,154.023
C07982=1071.646,-79.340,441.875,172.663,22.251,154.023
C07983=1071.640,-79.589,441.885,172.661,22.249,154.023
C07984=1071.633,-79.840,441.896,172.660,22.247,154.023
C07985=1071.627,-80.089,441.907,172.658,22.245,154.023
C07986=1071.622,-80.339,441.917,172.657,22.244,154.023
C07987=1071.615,-80.589,441.928,172.655,22.243,154.023
C07988=1071.609,-80.839,441.939,172.654,22.241,154.023
C07989=1071.603,-81.088,441.949,172.652,22.239,154.023
C07990=1071.597,-81.338,441.961,172.650,22.238,154.023
C07991=1071.590,-81.617,441.973,172.649,22.236,154.023
C07992=1071.583,-81.897,441.985,172.647,22.235,154.023
C07993=1071.576,-82.177,441.997,172.645,22.232,154.023
C07994=1071.569,-82.457,442.008,172.643,22.231,154.023
C07995=1071.563,-82.707,442.020,172.642,22.230,154.023
C07996=1071.557,-82.956,442.030,172.640,22.228,154.022
C07997=1071.551,-83.205,442.041,172.639,22.226,154.022
C07998=1071.545,-83.456,442.052,172.637,22.225,154.022
C07999=1071.539,-83.705,442.063,172.636,22.223,154.022
C08000=1071.532,-83.954,442.073,172.634,22.222,154.022
C08001=1071.526,-84.204,442.085,172.633,22.220,154.022
C08002=1071.521,-84.455,442.095,172.631,22.219,154.022
C08003=1071.514,-84.704,442.105,172.630,22.217,154.022
C08004=1071.508,-84.954,442.116,172.628,22.216,154.022
C08005=1071.501,-85.203,442.126,172.627,22.214,154.022
C08006=1071.496,-85.453,442.137,172.625,22.212,154.022
C08007=1071.489,-85.703,442.149,172.624,22.211,154.022
C08008=1071.483,-85.953,442.158,172.622,22.210,154.022
C08009=1071.477,-86.202,442.169,172.620,22.208,154.022
C08010=1071.472,-86.452,442.180,172.619,22.207,154.022
C08011=1071.464,-86.701,442.191,172.617,22.205,154.022
C08012=1071.459,-86.951,442.201,172.616,22.204,154.022
C08013=1071.453,-87.201,442.212,172.614,22.202,154.022
C08014=1071.447,-87.450,442.222,172.613,22.201,154.022
C08015=1071.440,-87.700,442.233,172.611,22.199,154.021
C08016=1071.435,-87.950,442.244,172.610,22.198,154.021
C08017=1071.428,-88.199,442.254,172.608,22.196,154.021
C08018=1071.423,-88.449,442.264,172.606,22.195,154.021
C08019=1071.416,-88.699,442.275,172.605,22.194,154.021
C08020=1071.410,-88.949,442.286,172.603,22.192,154.021
C08021=1071.405,-89.199,442.296,172.602,22.190,154.021
C08022=1071.398,-89.448,442.306,172.600,22.189,154.021
C08023=1071.392,-89.698,442.318,172.599,22.187,154.021
C08024=1071.385,-89.947,442.328,172.597,22.186,154.021
C08025=1071.380,-90.197,442.338,172.595,22.185,154.021
C08026=1071.374,-90.447,442.349,172.594,22.183,154.021
C08027=1071.368,-90.696,442.359,172.592,22.181,154.021
C08028=1071.362,-90.947,442.370,172.591,22.180,154.021
C08029=1071.355,-91.196,442.380,172.589,22.179,154.021
C08030=1071.349,-91.445,442.391,172.588,22.177,154.021
C08031=1071.344,-91.696,442.401,172.586,22.176,154.021
C08032=1071.337,-91.945,442.411,172.584,22.175,154.021
C08033=1071.331,-92.195,442.423,172.583,22.173,154.021
C08034=1071.325,-92.445,442.432,172.581,22.171,154.021
C08035=1071.319,-92.694,442.443,172.580,22.170,154.021
C08036=1071.313,-92.943,442.453,172.578,22.169,154.021
C08037=1071.307,-93.194,442.464,172.577,22.167,154.021
C08038=1071.302,-93.443,442.474,172.575,22.166,154.021
C08039=1071.295,-93.694,442.484,172.574,22.164,154.021
C08040=1071.289,-93.943,442.495,172.572,22.163,154.021
C08041=1071.283,-94.192,442.506,172.570,22.162,154.021
C08042=1071.277,-94.442,442.516,172.569,22.160,154.021
C08043=1071.271,-94.691,442.526,172.567,22.159,154.021
C08044=1071.265,-94.942,442.536,172.566,22.158,154.020
C08045=1071.259,-95.191,442.547,172.564,22.156,154.020
C08046=1071.253,-95.441,442.557,172.563,22.154,154.020
C08047=1071.247,-95.691,442.568,172.561,22.153,154.020
C08048=1071.241,-95.941,442.577,172.559,22.152,154.020
C08049=1071.235,-96.190,442.588,172.558,22.150,154.020
C08050=1071.229,-96.440,442.599,172.556,22.149,154.020
C08051=1071.223,-96.690,442.609,172.555,22.147,154.020
C08052=1071.217,-96.939,442.619,172.553,22.146,154.020
C08053=1071.211,-97.189,442.629,172.551,22.145,154.020
C08054=1071.205,-97.438,442.639,172.550,22.143,154.020
C08055=1071.198,-97.720,442.651,172.547,22.142,154.020
C08056=1071.192,-98.003,442.662,172.546,22.140,154.020
C08057=1071.184,-98.285,442.674,172.544,22.139,154.020
C08058=1071.177,-98.567,442.685,172.543,22.137,154.020
C08059=1071.171,-98.816,442.696,172.541,22.136,154.020
C08060=1071.165,-99.066,442.706,172.539,22.135,154.020
C08061=1071.158,-99.315,442.716,172.538,22.133,154.020
C08062=1071.153,-99.566,442.726,172.536,22.133,154.020
C08063=1071.147,-99.815,442.736,172.534,22.131,154.020
C08064=1071.140,-100.065,442.746,172.533,22.130,154.020
C08065=1071.135,-100.315,442.756,172.531,22.128,154.020
C08066=1071.128,-100.565,442.767,172.530,22.127,154.020
C08067=1071.122,-100.814,442.776,172.528,22.126,154.020
C08068=1071.116,-101.064,442.786,172.526,22.125,154.020
C08069=1071.110,-101.314,442.797,172.525,22.124,154.020
C08070=1071.104,-101.563,442.806,172.523,22.122,154.020
C08071=1071.098,-101.813,442.817,172.522,22.121,154.020
C08072=1071.092,-102.063,442.827,172.520,22.119,154.020
C08073=1071.085,-102.312,442.836,172.518,22.118,154.020
C08074=1071.079,-102.562,442.847,172.517,22.117,154.020
C08075=1071.074,-102.812,442.857,172.515,22.116,154.020
C08076=1071.067,-103.062,442.866,172.513,22.115,154.020
C08077=1071.061,-103.311,442.877,172.512,22.113,154.020
C08078=1071.055,-103.561,442.887,172.510,22.112,154.020
C08079=1071.049,-103.811,442.897,172.508,22.111,154.020
C08080=1071.042,-104.061,442.907,172.507,22.110,154.020
C08081=1071.036,-104.310,442.917,172.505,22.108,154.020
C08082=1071.031,-104.560,442.927,172.504,22.107,154.020
C08083=1071.024,-104.810,442.937,172.502,22.106,154.020
C08084=1071.018,-105.059,442.947,172.500,22.105,154.020
C08085=1071.012,-105.309,442.956,172.499,22.103,154.020
C08086=1071.006,-105.559,442.966,172.497,22.102,154.021
C08087=1071.000,-105.809,442.977,172.496,22.102,154.020
C08088=1070.994,-106.058,442.986,172.495,22.100,154.020
C08089=1070.988,-106.308,442.996,172.493,22.099,154.021
C08090=1070.982,-106.558,443.006,172.491,22.098,154.021
C08091=1070.976,-106.807,443.016,172.490,22.097,154.021
C08092=1070.969,-107.057,443.026,172.488,22.095,154.021
C08093=1070.963,-107.307,443.035,172.486,22.094,154.021
C08094=1070.957,-107.557,443.045,172.485,22.093,154.021
C08095=1070.951,-107.806,443.056,172.483,22.092,154.021
C08096=1070.945,-108.056,443.065,172.481,22.091,154.021
C08097=1070.939,-108.306,443.075,172.480,22.089,154.021
C08098=1070.933,-108.556,443.084,172.478,22.089,154.021
C08099=1070.927,-108.805,443.094,172.476,22.087,154.021
C08100=1070.921,-109.055,443.104,172.475,22.086,154.021
C08101=1070.914,-109.304,443.114,172.473,22.085,154.021
C08102=1070.908,-109.554,443.123,172.471,22.084,154.021
C08103=1070.902,-109.804,443.133,172.470,22.083,154.021
C08104=1070.896,-110.054,443.143,172.468,22.082,154.021
C08105=1070.890,-110.304,443.153,172.466,22.081,154.021
C08106=1070.884,-110.554,443.162,172.465,22.079,154.021
C08107=1070.877,-110.803,443.173,172.463,22.079,154.021
C08108=1070.871,-111.053,443.182,172.461,22.077,154.021
C08109=1070.865,-111.303,443.192,172.460,22.077,154.021
C08110=1070.859,-111.552,443.201,172.459,22.075,154.021
C08111=1070.853,-111.802,443.211,172.457,22.075,154.021
C08112=1070.847,-112.052,443.220,172.456,22.073,154.021
C08113=1070.840,-112.302,443.230,172.454,22.072,154.021
C08114=1070.834,-112.552,443.240,172.452,22.071,154.021
C08115=1070.828,-112.801,443.249,172.451,22.070,154.021
C08116=1070.823,-113.051,443.259,172.449,22.069,154.022
C08117=1070.816,-113.301,443.269,172.447,22.067,154.022
C08118=1070.811,-113.550,443.278,172.445,22.067,154.022
C08119=1070.803,-113.829,443.289,172.444,22.065,154.022
C08120=1070.796,-114.110,443.300,172.442,22.064,154.022
C08121=1070.790,-114.390,443.311,172.440,22.063,154.022
C08122=1070.783,-114.669,443.321,172.438,22.062,154.022
C08123=1070.776,-114.919,443.331,172.436,22.061,154.022
C08124=1070.770,-115.168,443.341,172.434,22.060,154.022
C08125=1070.765,-115.417,443.350,172.434,22.059,154.022
C08126=1070.758,-115.667,443.359,172.432,22.058,154.022
C08127=1070.752,-115.917,443.369,172.430,22.057,154.022
C08128=1070.746,-116.167,443.379,172.428,22.056,154.022
C08129=1070.740,-116.417,443.388,172.427,22.055,154.022
C08130=1070.734,-116.666,443.398,172.425,22.054,154.022
C08131=1070.728,-116.916,443.407,172.423,22.053,154.022
C08132=1070.721,-117.166,443.417,172.422,22.052,154.022
C08133=1070.715,-117.416,443.426,172.420,22.051,154.023
C08134=1070.709,-117.666,443.436,172.418,22.050,154.023
C08135=1070.703,-117.916,443.445,172.416,22.049,154.023
C08136=1070.698,-118.165,443.454,172.415,22.048,154.023
C08137=1070.691,-118.415,443.463,172.413,22.047,154.023
C08138=1070.685,-118.664,443.473,172.411,22.046,154.023
C08139=1070.678,-118.914,443.482,172.410,22.046,154.023
C08140=1070.672,-119.164,443.492,172.409,22.045,154.023
C08141=1070.666,-119.414,443.501,172.407,22.043,154.023
C08142=1070.660,-119.664,443.511,172.405,22.043,154.023
C08143=1070.654,-119.913,443.520,172.404,22.042,154.023
C08144=1070.648,-120.163,443.530,172.402,22.041,154.023
C08145=1070.642,-120.413,443.538,172.400,22.040,154.023
C08146=1070.635,-120.662,443.547,172.398,22.039,154.024
C08147=1070.629,-120.912,443.557,172.397,22.038,154.024
C08148=1070.623,-121.162,443.567,172.395,22.037,154.024
C08149=1070.617,-121.412,443.576,172.393,22.036,154.024
C08150=1070.611,-121.662,443.586,172.391,22.035,154.024
C08151=1070.605,-121.911,443.595,172.391,22.035,154.024
C08152=1070.599,-122.161,443.604,172.389,22.034,154.024
C08153=1070.592,-122.411,443.613,172.387,22.032,154.024
C08154=1070.586,-122.660,443.622,172.385,22.032,154.024
C08155=1070.580,-122.910,443.632,172.384,22.031,154.024
C08156=1070.574,-123.160,443.641,172.382,22.030,154.024
C08157=1070.569,-123.410,443.650,172.380,22.029,154.024
C08158=1070.562,-123.660,443.659,172.378,22.028,154.025
C08159=1070.555,-123.909,443.668,172.377,22.027,154.025
C08160=1070.549,-124.159,443.678,172.375,22.026,154.025
C08161=1070.543,-124.409,443.687,172.373,22.025,154.025
C08162=1070.537,-124.659,443.696,172.372,22.025,154.025
C08163=1070.532,-124.908,443.706,172.370,22.024,154.025
C08164=1070.525,-125.158,443.715,172.369,22.023,154.025
C08165=1070.519,-125.408,443.723,172.367,22.022,154.025
C08166=1070.513,-125.658,443.733,172.365,22.022,154.025
C08167=1070.507,-125.908,443.743,172.363,22.021,154.025
C08168=1070.500,-126.156,443.751,172.362,22.019,154.025
C08169=1070.494,-126.407,443.760,172.360,22.019,154.026
C08170=1070.488,-126.657,443.770,172.358,22.018,154.026
C08171=1070.481,-126.906,443.779,172.356,22.017,154.026
C08172=1070.475,-127.157,443.787,172.356,22.017,154.026
C08173=1070.470,-127.406,443.797,172.354,22.016,154.026
C08174=1070.464,-127.655,443.806,172.352,22.015,154.026
C08175=1070.457,-127.907,443.815,172.350,22.014,154.026
C08176=1070.452,-128.157,443.825,172.349,22.013,154.026
C08177=1070.450,-128.408,443.836,172.347,22.011,154.026
C08178=1070.449,-128.658,443.846,172.346,22.008,154.026
C08179=1070.451,-128.911,443.860,172.345,22.005,154.025
C08180=1070.454,-129.164,443.873,172.345,22.001,154.025
C08181=1070.459,-129.416,443.886,172.344,21.995,154.024
C08182=1070.467,-129.666,443.901,172.344,21.990,154.023
C08183=1070.077,-129.688,443.736,172.298,22.130,154.055
C08184=1070.069,-129.439,443.720,172.298,22.135,154.056
C08185=1070.063,-129.187,443.706,172.299,22.140,154.057
C08186=1070.060,-128.934,443.693,172.299,22.145,154.057
C08187=1070.059,-128.681,443.680,172.300,22.148,154.058
C08188=1070.060,-128.430,443.669,172.300,22.150,154.058
C08189=1070.062,-128.180,443.659,172.302,22.153,154.059
C08190=1070.066,-127.929,443.649,172.303,22.154,154.059
C08191=1070.073,-127.678,443.640,172.305,22.155,154.058
C08192=1070.079,-127.428,443.630,172.307,22.156,154.058
C08193=1070.084,-127.178,443.621,172.309,22.157,154.058
C08194=1070.091,-126.929,443.612,172.310,22.157,154.058
C08195=1070.097,-126.679,443.603,172.312,22.158,154.058
C08196=1070.104,-126.429,443.593,172.314,22.159,154.058
C08197=1070.109,-126.180,443.585,172.316,22.160,154.058
C08198=1070.116,-125.930,443.576,172.317,22.160,154.058
C08199=1070.122,-125.680,443.566,172.318,22.161,154.058
C08200=1070.128,-125.430,443.557,172.320,22.162,154.057
C08201=1070.134,-125.180,443.548,172.322,22.163,154.057
C08202=1070.141,-124.931,443.539,172.324,22.164,154.057
C08203=1070.146,-124.681,443.530,172.325,22.165,154.057
C08204=1070.152,-124.431,443.521,172.327,22.166,154.057
C08205=1070.158,-124.181,443.511,172.329,22.166,154.057
C08206=1070.165,-123.932,443.502,172.331,22.167,154.057
C08207=1070.171,-123.682,443.493,172.332,22.168,154.057
C08208=1070.180,-123.325,443.480,172.334,22.169,154.057
C08209=1070.188,-122.968,443.466,172.337,22.171,154.057
C08210=1070.197,-122.610,443.453,172.339,22.172,154.056
C08211=1070.206,-122.253,443.440,172.342,22.173,154.056
C08212=1070.212,-122.003,443.430,172.344,22.174,154.056
C08213=1070.218,-121.754,443.421,172.345,22.175,154.056
C08214=1070.224,-121.504,443.413,172.346,22.176,154.056
C08215=1070.231,-121.254,443.403,172.348,22.176,154.056
C08216=1070.237,-121.005,443.394,172.350,22.178,154.056
C08217=1070.243,-120.755,443.384,172.352,22.179,154.056
C08218=1070.249,-120.505,443.375,172.353,22.179,154.056
C08219=1070.255,-120.255,443.365,172.355,22.180,154.056
C08220=1070.261,-120.005,443.355,172.357,22.182,154.056
C08221=1070.267,-119.756,443.347,172.358,22.182,154.056
C08222=1070.274,-119.506,443.338,172.360,22.183,154.055
C08223=1070.280,-119.256,443.328,172.362,22.184,154.055
C08224=1070.286,-119.007,443.319,172.364,22.185,154.055
C08225=1070.292,-118.757,443.309,172.365,22.186,154.055
C08226=1070.298,-118.507,443.300,172.366,22.187,154.055
C08227=1070.304,-118.257,443.290,172.368,22.188,154.055
C08228=1070.311,-118.007,443.281,172.370,22.189,154.055
C08229=1070.317,-117.758,443.271,172.371,22.190,154.055
C08230=1070.322,-117.509,443.262,172.373,22.191,154.055
C08231=1070.329,-117.259,443.252,172.375,22.192,154.055
C08232=1070.335,-117.009,443.243,172.377,22.192,154.055
C08233=1070.341,-116.759,443.234,172.378,22.194,154.055
C08234=1070.347,-116.509,443.224,172.380,22.195,154.055
C08235=1070.353,-116.259,443.215,172.382,22.196,154.055
C08236=1070.359,-116.009,443.205,172.383,22.197,154.054
C08237=1070.366,-115.760,443.196,172.385,22.198,154.054
C08238=1070.372,-115.510,443.187,172.387,22.199,154.054
C08239=1070.378,-115.260,443.177,172.389,22.200,154.054
C08240=1070.388,-114.838,443.161,172.391,22.202,154.054
C08241=1070.399,-114.416,443.144,172.394,22.203,154.054
C08242=1070.409,-113.994,443.128,172.396,22.205,154.054
C08243=1070.420,-113.572,443.112,172.400,22.207,154.054
C08244=1070.426,-113.322,443.103,172.401,22.208,154.054
C08245=1070.432,-113.072,443.093,172.403,22.209,154.054
C08246=1070.438,-112.822,443.083,172.405,22.210,154.054
C08247=1070.444,-112.573,443.073,172.405,22.211,154.054
C08248=1070.450,-112.323,443.064,172.407,22.212,154.054
C08249=1070.456,-112.073,443.054,172.409,22.213,154.054
C08250=1070.463,-111.824,443.044,172.410,22.214,154.054
C08251=1070.469,-111.574,443.034,172.412,22.215,154.054
C08252=1070.474,-111.325,443.025,172.414,22.216,154.054
C08253=1070.480,-111.075,443.016,172.416,22.217,154.053
C08254=1070.487,-110.825,443.006,172.417,22.219,154.053
C08255=1070.493,-110.576,442.996,172.419,22.219,154.053
C08256=1070.499,-110.326,442.987,172.421,22.221,154.053
C08257=1070.505,-110.076,442.977,172.422,22.221,154.053
C08258=1070.511,-109.826,442.966,172.424,22.223,154.053
C08259=1070.517,-109.577,442.957,172.426,22.224,154.053
C08260=1070.523,-109.327,442.947,172.427,22.225,154.053
C08261=1070.529,-109.077,442.938,172.429,22.226,154.053
C08262=1070.536,-108.827,442.928,172.431,22.227,154.053
C08263=1070.542,-108.577,442.919,172.432,22.229,154.053
C08264=1070.548,-108.328,442.908,172.434,22.230,154.053
C08265=1070.554,-108.078,442.899,172.436,22.231,154.053
C08266=1070.561,-107.829,442.889,172.437,22.232,154.053
C08267=1070.566,-107.579,442.879,172.439,22.233,154.053
C08268=1070.573,-107.328,442.869,172.440,22.234,154.053
C08269=1070.579,-107.079,442.859,172.441,22.235,154.053
C08270=1070.585,-106.829,442.849,172.443,22.236,154.053
C08271=1070.592,-106.579,442.840,172.445,22.237,154.053
C08272=1070.597,-106.329,442.829,172.446,22.239,154.053
C08273=1070.603,-106.080,442.819,172.448,22.240,154.053
C08274=1070.610,-105.830,442.810,172.450,22.241,154.053
C08275=1070.616,-105.580,442.800,172.451,22.242,154.053
C08276=1070.621,-105.330,442.790,172.453,22.244,154.053
C08277=1070.628,-105.081,442.780,172.455,22.244,154.053
C08278=1070.634,-104.831,442.770,172.456,22.246,154.053
C08279=1070.640,-104.582,442.760,172.458,22.247,154.053
C08280=1070.646,-104.332,442.750,172.459,22.249,154.053
C08281=1070.652,-104.082,442.740,172.461,22.249,154.053
C08282=1070.658,-103.832,442.730,172.463,22.251,154.053
C08283=1070.665,-103.583,442.720,172.464,22.252,154.053
C08284=1070.670,-103.333,442.710,172.466,22.253,154.053
C08285=1070.676,-103.083,442.700,172.468,22.254,154.053
C08286=1070.683,-102.834,442.690,172.469,22.256,154.053
C08287=1070.688,-102.584,442.680,172.471,22.257,154.053
C08288=1070.694,-102.334,442.670,172.473,22.258,154.053
C08289=1070.701,-102.085,442.660,172.474,22.260,154.053
C08290=1070.706,-101.835,442.650,172.476,22.261,154.053
C08291=1070.713,-101.584,442.640,172.478,22.262,154.053
C08292=1070.719,-101.335,442.630,172.479,22.263,154.053
C08293=1070.726,-101.085,442.620,172.481,22.265,154.053
C08294=1070.731,-100.836,442.609,172.482,22.266,154.053
C08295=1070.738,-100.586,442.600,172.484,22.267,154.053
C08296=1070.744,-100.336,442.590,172.486,22.269,154.053
C08297=1070.749,-100.087,442.579,172.487,22.269,154.052
C08298=1070.756,-99.837,442.570,172.489,22.271,154.053
C08299=1070.762,-99.588,442.559,172.491,22.272,154.053
C08300=1070.768,-99.338,442.549,172.492,22.274,154.053
C08301=1070.775,-99.088,442.539,172.494,22.275,154.053
C08302=1070.781,-98.838,442.529,172.495,22.276,154.053
C08303=1070.786,-98.588,442.519,172.497,22.278,154.053
C08304=1070.793,-98.306,442.507,172.499,22.279,154.053
C08305=1070.800,-98.024,442.496,172.500,22.280,154.053
C08306=1070.807,-97.742,442.485,172.502,22.282,154.053
C08307=1070.814,-97.461,442.473,172.504,22.284,154.053
C08308=1070.821,-97.210,442.463,172.506,22.285,154.053
C08309=1070.826,-96.961,442.452,172.507,22.286,154.053
C08310=1070.833,-96.711,442.442,172.508,22.287,154.053
C08311=1070.838,-96.461,442.432,172.510,22.289,154.053
C08312=1070.844,-96.211,442.421,172.511,22.290,154.053
C08313=1070.850,-95.962,442.411,172.513,22.291,154.053
C08314=1070.856,-95.712,442.401,172.514,22.293,154.053
C08315=1070.862,-95.463,442.391,172.516,22.294,154.053
C08316=1070.868,-95.213,442.380,172.518,22.295,154.053
C08317=1070.875,-94.963,442.370,172.519,22.297,154.053
C08318=1070.880,-94.713,442.359,172.521,22.298,154.053
C08319=1070.887,-94.463,442.349,172.522,22.299,154.053
C08320=1070.892,-94.214,442.339,172.524,22.301,154.053
C08321=1070.898,-93.964,442.329,172.525,22.303,154.053
C08322=1070.904,-93.715,442.318,172.527,22.304,154.053
C08323=1070.910,-93.465,442.307,172.529,22.305,154.053
C08324=1070.917,-93.215,442.297,172.530,22.307,154.053
C08325=1070.922,-92.965,442.286,172.532,22.308,154.053
C08326=1070.929,-92.716,442.276,172.533,22.310,154.053
C08327=1070.934,-92.466,442.266,172.535,22.311,154.053
C08328=1070.941,-92.217,442.256,172.537,22.312,154.053
C08329=1070.946,-91.967,442.245,172.538,22.314,154.053
C08330=1070.953,-91.716,442.234,172.540,22.316,154.053
C08331=1070.959,-91.467,442.224,172.541,22.317,154.053
C08332=1070.965,-91.217,442.214,172.543,22.318,154.053
C08333=1070.971,-90.968,442.204,172.544,22.320,154.053
C08334=1070.977,-90.718,442.193,172.546,22.321,154.053
C08335=1070.983,-90.468,442.182,172.548,22.322,154.053
C08336=1070.989,-90.218,442.172,172.549,22.324,154.054
C08337=1070.995,-89.969,442.161,172.551,22.326,154.054
C08338=1071.001,-89.720,442.151,172.552,22.327,154.054
C08339=1071.007,-89.470,442.141,172.554,22.328,154.054
C08340=1071.013,-89.219,442.129,172.556,22.330,154.054
C08341=1071.020,-88.970,442.119,172.558,22.331,154.054
C08342=1071.025,-88.721,442.108,172.559,22.333,154.054
C08343=1071.032,-88.471,442.099,172.561,22.335,154.054
C08344=1071.038,-88.221,442.087,172.563,22.336,154.054
C08345=1071.044,-87.971,442.076,172.564,22.337,154.054
C08346=1071.050,-87.722,442.066,172.566,22.339,154.054
C08347=1071.056,-87.472,442.056,172.567,22.341,154.054
C08348=1071.062,-87.222,442.045,172.569,22.342,154.054
C08349=1071.068,-86.973,442.034,172.570,22.343,154.054
C08350=1071.074,-86.723,442.024,172.572,22.345,154.054
C08351=1071.080,-86.473,442.013,172.573,22.347,154.054
C08352=1071.087,-86.223,442.003,172.575,22.348,154.054
C08353=1071.092,-85.974,441.992,172.577,22.349,154.054
C08354=1071.099,-85.724,441.982,172.578,22.351,154.054
C08355=1071.105,-85.474,441.970,172.580,22.353,154.054
C08356=1071.111,-85.225,441.959,172.581,22.354,154.054
C08357=1071.117,-84.975,441.950,172.583,22.355,154.054
C08358=1071.124,-84.725,441.939,172.584,22.357,154.054
C08359=1071.129,-84.475,441.928,172.586,22.359,154.055
C08360=1071.136,-84.226,441.918,172.587,22.360,154.055
C08361=1071.141,-83.977,441.907,172.589,22.361,154.055
C08362=1071.148,-83.726,441.895,172.590,22.363,154.055
C08363=1071.154,-83.477,441.885,172.592,22.365,154.055
C08364=1071.160,-83.228,441.874,172.594,22.366,154.055
C08365=1071.166,-82.977,441.864,172.595,22.367,154.055
C08366=1071.173,-82.728,441.853,172.597,22.369,154.055
C08367=1071.178,-82.478,441.843,172.598,22.371,154.055
C08368=1071.185,-82.198,441.830,172.600,22.373,154.055
C08369=1071.193,-81.919,441.818,172.602,22.374,154.055
C08370=1071.200,-81.639,441.806,172.603,22.376,154.055
C08371=1071.206,-81.359,441.794,172.605,22.378,154.055
C08372=1071.212,-81.109,441.783,172.607,22.379,154.055
C08373=1071.219,-80.860,441.772,172.608,22.381,154.055
C08374=1071.225,-80.609,441.761,172.610,22.382,154.055
C08375=1071.231,-80.360,441.750,172.611,22.384,154.055
C08376=1071.237,-80.111,441.740,172.613,22.386,154.056
C08377=1071.244,-79.861,441.729,172.614,22.387,154.056
C08378=1071.249,-79.611,441.718,172.616,22.389,154.056
C08379=1071.255,-79.362,441.707,172.617,22.390,154.056
C08380=1071.261,-79.111,441.696,172.619,22.392,154.056
C08381=1071.267,-78.862,441.685,172.620,22.394,154.056
C08382=1071.273,-78.612,441.674,172.622,22.395,154.056
C08383=1071.280,-78.363,441.663,172.623,22.397,154.056
C08384=1071.286,-78.113,441.652,172.625,22.399,154.056
C08385=1071.291,-77.864,441.642,172.626,22.400,154.056
C08386=1071.298,-77.613,441.630,172.629,22.402,154.056
C08387=1071.303,-77.364,441.619,172.630,22.404,154.056
C08388=1071.310,-77.114,441.608,172.632,22.406,154.056
C08389=1071.316,-76.864,441.597,172.633,22.407,154.057
C08390=1071.321,-76.615,441.586,172.635,22.409,154.057
C08391=1071.328,-76.365,441.575,172.636,22.410,154.057
C08392=1071.334,-76.116,441.564,172.638,22.412,154.057
C08393=1071.340,-75.866,441.552,172.639,22.414,154.057
C08394=1071.346,-75.616,441.542,172.641,22.415,154.057
C08395=1071.352,-75.367,441.531,172.642,22.417,154.057
C08396=1071.359,-75.117,441.520,172.644,22.419,154.057
C08397=1071.364,-74.867,441.509,172.645,22.420,154.057
C08398=1071.371,-74.617,441.498,172.647,22.422,154.057
C08399=1071.376,-74.367,441.487,172.648,22.424,154.057
C08400=1071.382,-74.119,441.475,172.650,22.425,154.057
C08401=1071.389,-73.868,441.464,172.651,22.427,154.058
C08402=1071.395,-73.619,441.453,172.653,22.429,154.058
C08403=1071.401,-73.369,441.442,172.654,22.430,154.058
C08404=1071.407,-73.119,441.431,172.656,22.432,154.058
C08405=1071.412,-72.869,441.420,172.657,22.434,154.058
C08406=1071.418,-72.620,441.408,172.659,22.436,154.058
C08407=1071.424,-72.370,441.397,172.660,22.438,154.058
C08408=1071.430,-72.121,441.386,172.661,22.439,154.058
C08409=1071.436,-71.871,441.375,172.663,22.441,154.058
C08410=1071.442,-71.622,441.363,172.665,22.443,154.059
C08411=1071.448,-71.372,441.352,172.667,22.445,154.059
C08412=1071.453,-71.122,441.340,172.668,22.447,154.059
C08413=1071.459,-70.872,441.329,172.670,22.448,154.059
C08414=1071.466,-70.623,441.318,172.671,22.450,154.059
C08415=1071.472,-70.373,441.307,172.673,22.452,154.059
C08416=1071.478,-70.123,441.295,172.674,22.454,154.059
C08417=1071.484,-69.874,441.285,172.676,22.455,154.059
C08418=1071.490,-69.624,441.272,172.677,22.457,154.059
C08419=1071.495,-69.374,441.261,172.678,22.459,154.060
C08420=1071.501,-69.125,441.250,172.680,22.461,154.060
C08421=1071.508,-68.875,441.238,172.682,22.463,154.060
C08422=1071.513,-68.626,441.227,172.683,22.464,154.060
C08423=1071.519,-68.375,441.216,172.684,22.466,154.060
C08424=1071.525,-68.126,441.205,172.686,22.468,154.060
C08425=1071.531,-67.876,441.193,172.687,22.470,154.060
C08426=1071.537,-67.627,441.182,172.689,22.472,154.060
C08427=1071.544,-67.377,441.170,172.690,22.473,154.061
C08428=1071.549,-67.127,441.158,172.692,22.475,154.061
C08429=1071.555,-66.877,441.147,172.693,22.477,154.061
C08430=1071.561,-66.628,441.136,172.695,22.480,154.061
C08431=1071.568,-66.378,441.124,172.697,22.481,154.061
C08432=1071.574,-66.101,441.112,172.698,22.483,154.061
C08433=1071.580,-65.823,441.099,172.700,22.485,154.061
C08434=1071.587,-65.546,441.086,172.701,22.487,154.062
C08435=1071.594,-65.268,441.073,172.703,22.489,154.062
C08436=1071.599,-65.018,441.062,172.705,22.491,154.062
C08437=1071.606,-64.768,441.050,172.706,22.493,154.062
C08438=1071.612,-64.519,441.039,172.708,22.495,154.062
C08439=1071.618,-64.269,441.027,172.709,22.497,154.062
C08440=1071.623,-64.019,441.016,172.711,22.498,154.062
C08441=1071.630,-63.770,441.004,172.712,22.500,154.062
C08442=1071.636,-63.520,440.993,172.713,22.502,154.063
C08443=1071.642,-63.270,440.982,172.715,22.504,154.063
C08444=1071.648,-63.021,440.970,172.716,22.506,154.063
C08445=1071.654,-62.771,440.958,172.718,22.507,154.063
C08446=1071.660,-62.521,440.946,172.719,22.509,154.063
C08447=1071.666,-62.272,440.935,172.721,22.511,154.063
C08448=1071.673,-62.022,440.923,172.723,22.514,154.063
C08449=1071.678,-61.772,440.912,172.724,22.516,154.063
C08450=1071.684,-61.523,440.900,172.726,22.517,154.064
C08451=1071.690,-61.273,440.889,172.727,22.519,154.064
C08452=1071.696,-61.023,440.876,172.729,22.521,154.064
C08453=1071.703,-60.774,440.865,172.730,22.523,154.064
C08454=1071.709,-60.524,440.854,172.732,22.525,154.064
C08455=1071.715,-60.275,440.842,172.733,22.526,154.064
C08456=1071.720,-60.025,440.830,172.735,22.528,154.064
C08457=1071.727,-59.775,440.818,172.736,22.530,154.064
C08458=1071.733,-59.525,440.807,172.737,22.532,154.065
C08459=1071.738,-59.276,440.795,172.739,22.534,154.065
C08460=1071.745,-59.027,440.783,172.740,22.536,154.065
C08461=1071.751,-58.777,440.772,172.742,22.538,154.065
C08462=1071.757,-58.527,440.760,172.743,22.540,154.065
C08463=1071.763,-58.277,440.748,172.746,22.542,154.065
C08464=1071.769,-58.028,440.737,172.747,22.543,154.065
C08465=1071.776,-57.779,440.725,172.748,22.545,154.066
C08466=1071.781,-57.528,440.713,172.750,22.547,154.066
C08467=1071.787,-57.279,440.701,172.751,22.549,154.066
C08468=1071.794,-57.030,440.689,172.753,22.551,154.066
C08469=1071.800,-56.779,440.677,172.754,22.553,154.066
C08470=1071.806,-56.530,440.666,172.756,22.555,154.066
C08471=1071.812,-56.281,440.654,172.757,22.557,154.066
C08472=1071.819,-56.030,440.643,172.758,22.559,154.067
C08473=1071.824,-55.781,440.630,172.760,22.561,154.067
C08474=1071.831,-55.532,440.618,172.761,22.562,154.067
C08475=1071.837,-55.281,440.607,172.763,22.564,154.067
C08476=1071.842,-55.032,440.595,172.764,22.566,154.067
C08477=1071.849,-54.783,440.583,172.766,22.569,154.067
C08478=1071.855,-54.533,440.572,172.768,22.571,154.067
C08479=1071.861,-54.283,440.559,172.769,22.572,154.068
C08480=1071.867,-54.034,440.548,172.771,22.574,154.068
C08481=1071.873,-53.784,440.535,172.772,22.576,154.068
C08482=1071.879,-53.534,440.524,172.773,22.578,154.068
C08483=1071.886,-53.285,440.512,172.775,22.580,154.068
C08484=1071.891,-53.035,440.500,172.776,22.582,154.068
C08485=1071.898,-52.785,440.488,172.778,22.584,154.068
C08486=1071.905,-52.536,440.476,172.779,22.586,154.069
C08487=1071.910,-52.286,440.464,172.781,22.588,154.069
C08488=1071.916,-52.036,440.452,172.782,22.590,154.069
C08489=1071.923,-51.787,440.440,172.783,22.591,154.069
C08490=1071.929,-51.537,440.428,172.786,22.594,154.069
C08491=1071.935,-51.288,440.416,172.787,22.596,154.069
C08492=1071.941,-51.038,440.404,172.789,22.598,154.069
C08493=1071.947,-50.788,440.392,172.790,22.599,154.070
C08494=1071.954,-50.538,440.381,172.791,22.601,154.070
C08495=1071.959,-50.289,440.368,172.793,22.603,154.070
C08496=1071.966,-50.013,440.355,172.794,22.606,154.070
C08497=1071.973,-49.736,440.341,172.796,22.608,154.070
C08498=1071.979,-49.460,440.328,172.798,22.611,154.071
C08499=1071.986,-49.184,440.315,172.799,22.612,154.071
C08500=1071.992,-48.934,440.302,172.801,22.614,154.071
C08501=1071.998,-48.685,440.290,172.802,22.617,154.071
C08502=1072.004,-48.435,440.278,172.803,22.619,154.071
C08503=1072.009,-48.185,440.266,172.805,22.621,154.071
C08504=1072.015,-47.935,440.254,172.807,22.623,154.072
C08505=1072.022,-47.686,440.242,172.808,22.625,154.072
C08506=1072.028,-47.436,440.229,172.810,22.627,154.072
C08507=1072.033,-47.187,440.217,172.811,22.629,154.072
C08508=1072.040,-46.937,440.205,172.812,22.631,154.072
C08509=1072.046,-46.687,440.193,172.814,22.634,154.073
C08510=1072.051,-46.437,440.180,172.815,22.635,154.073
C08511=1072.058,-46.188,440.168,172.817,22.637,154.073
C08512=1072.063,-45.939,440.156,172.818,22.639,154.073
C08513=1072.069,-45.689,440.143,172.819,22.642,154.073
C08514=1072.076,-45.439,440.131,172.821,22.644,154.073
C08515=1072.081,-45.190,440.119,172.822,22.645,154.074
C08516=1072.087,-44.940,440.107,172.824,22.648,154.074
C08517=1072.094,-44.690,440.095,172.826,22.650,154.074
C08518=1072.100,-44.441,440.082,172.827,22.652,154.074
C08519=1072.106,-44.191,440.070,172.828,22.654,154.074
C08520=1072.112,-43.942,440.058,172.830,22.656,154.074
C08521=1072.118,-43.692,440.045,172.831,22.658,154.075
C08522=1072.124,-43.442,440.033,172.833,22.660,154.075
C08523=1072.129,-43.192,440.020,172.834,22.662,154.075
C08524=1072.136,-42.943,440.008,172.835,22.665,154.075
C08525=1072.141,-42.693,439.996,172.837,22.667,154.075
C08526=1072.147,-42.443,439.984,172.838,22.668,154.076
C08527=1072.154,-42.195,439.971,172.840,22.671,154.076
C08528=1072.160,-41.945,439.958,172.842,22.673,154.076
C08529=1072.166,-41.695,439.946,172.843,22.675,154.076
C08530=1072.172,-41.445,439.933,172.845,22.677,154.076
C08531=1072.178,-41.196,439.922,172.846,22.679,154.077
C08532=1072.184,-40.946,439.909,172.847,22.681,154.077
C08533=1072.190,-40.696,439.897,172.849,22.683,154.077
C08534=1072.196,-40.447,439.885,172.850,22.686,154.077
C08535=1072.203,-40.197,439.871,172.851,22.688,154.077
C08536=1072.209,-39.948,439.859,172.853,22.690,154.077
C08537=1072.215,-39.698,439.846,172.854,22.692,154.078
C08538=1072.221,-39.449,439.835,172.855,22.694,154.078
C08539=1072.226,-39.199,439.822,172.858,22.696,154.078
C08540=1072.232,-38.949,439.810,172.859,22.699,154.078
C08541=1072.239,-38.700,439.796,172.860,22.701,154.078
C08542=1072.244,-38.450,439.784,172.862,22.702,154.079
C08543=1072.250,-38.200,439.771,172.863,22.705,154.079
C08544=1072.257,-37.950,439.759,172.864,22.707,154.079
C08545=1072.263,-37.701,439.747,172.866,22.709,154.079
C08546=1072.269,-37.452,439.734,172.867,22.711,154.079
C08547=1072.274,-37.202,439.721,172.868,22.714,154.080
C08548=1072.280,-36.952,439.709,172.870,22.715,154.080
C08549=1072.286,-36.702,439.696,172.872,22.718,154.080
C08550=1072.293,-36.453,439.683,172.873,22.720,154.080
C08551=1072.298,-36.203,439.670,172.875,22.722,154.080
C08552=1072.304,-35.953,439.658,172.876,22.725,154.081
C08553=1072.310,-35.704,439.646,172.878,22.726,154.081
C08554=1072.316,-35.455,439.632,172.879,22.729,154.081
C08555=1072.322,-35.205,439.620,172.880,22.731,154.081
C08556=1072.328,-34.955,439.607,172.881,22.733,154.082
C08557=1072.334,-34.706,439.594,172.883,22.735,154.082
C08558=1072.340,-34.456,439.581,172.884,22.738,154.082
C08559=1072.346,-34.206,439.569,172.886,22.739,154.082
C08560=1072.352,-33.931,439.555,172.888,22.742,154.082
C08561=1072.359,-33.654,439.541,172.889,22.745,154.083
C08562=1072.365,-33.379,439.527,172.890,22.747,154.083
C08563=1072.372,-33.103,439.513,172.893,22.750,154.083
C08564=1072.379,-32.853,439.499,172.894,22.752,154.083
C08565=1072.385,-32.603,439.487,172.895,22.754,154.084
C08566=1072.390,-32.354,439.474,172.896,22.756,154.084
C08567=1072.397,-32.104,439.461,172.898,22.758,154.084
C08568=1072.403,-31.854,439.448,172.899,22.761,154.084
C08569=1072.409,-31.605,439.435,172.901,22.763,154.084
C08570=1072.415,-31.355,439.423,172.902,22.765,154.085
C08571=1072.420,-31.106,439.410,172.904,22.767,154.085
C08572=1072.426,-30.857,439.397,172.905,22.770,154.085
C08573=1072.432,-30.607,439.385,172.907,22.772,154.085
C08574=1072.438,-30.358,439.371,172.908,22.774,154.085
C08575=1072.444,-30.108,439.359,172.910,22.776,154.086
C08576=1072.451,-29.859,439.346,172.911,22.778,154.086
C08577=1072.456,-29.609,439.333,172.912,22.780,154.086
C08578=1072.463,-29.359,439.320,172.913,22.783,154.086
C08579=1072.469,-29.110,439.307,172.915,22.785,154.087
C08580=1072.474,-28.860,439.295,172.916,22.787,154.087
C08581=1072.481,-28.610,439.281,172.918,22.790,154.087
C08582=1072.487,-28.360,439.269,172.920,22.792,154.087
C08583=1072.493,-28.111,439.256,172.921,22.794,154.087
C08584=1072.499,-27.862,439.242,172.922,22.796,154.088
C08585=1072.504,-27.612,439.229,172.924,22.799,154.088
C08586=1072.510,-27.362,439.216,172.925,22.801,154.088
C08587=1072.517,-27.112,439.203,172.926,22.803,154.088
C08588=1072.523,-26.863,439.190,172.928,22.805,154.088
C08589=1072.529,-26.613,439.177,172.929,22.807,154.089
C08590=1072.535,-26.363,439.164,172.930,22.810,154.089
C08591=1072.541,-26.114,439.151,172.933,22.812,154.089
C08592=1072.547,-25.864,439.137,172.934,22.814,154.089
C08593=1072.553,-25.614,439.125,172.935,22.817,154.090
C08594=1072.559,-25.365,439.112,172.937,22.819,154.090
C08595=1072.565,-25.116,439.098,172.938,22.821,154.090
C08596=1072.570,-24.865,439.085,172.939,22.824,154.090
C08597=1072.576,-24.616,439.072,172.941,22.826,154.091
C08598=1072.583,-24.367,439.059,172.942,22.828,154.091
C08599=1072.588,-24.117,439.046,172.943,22.830,154.091
C08600=1072.595,-23.868,439.033,172.944,22.832,154.091
C08601=1072.600,-23.618,439.020,172.947,22.835,154.092
C08602=1072.606,-23.368,439.006,172.948,22.838,154.092
C08603=1072.612,-23.119,438.993,172.949,22.840,154.092
C08604=1072.617,-22.869,438.980,172.951,22.842,154.092
C08605=1072.624,-22.620,438.967,172.952,22.844,154.093
C08606=1072.630,-22.370,438.953,172.953,22.846,154.093
C08607=1072.636,-22.120,438.941,172.955,22.849,154.093
C08608=1072.641,-21.871,438.927,172.956,22.851,154.093
C08609=1072.647,-21.622,438.914,172.957,22.853,154.093
C08610=1072.654,-21.372,438.900,172.959,22.856,154.094
C08611=1072.660,-21.122,438.888,172.961,22.858,154.094
C08612=1072.665,-20.873,438.874,172.962,22.861,154.094
C08613=1072.671,-20.624,438.861,172.963,22.863,154.094
C08614=1072.677,-20.374,438.848,172.965,22.865,154.095
C08615=1072.683,-20.123,438.834,172.966,22.868,154.095
C08616=1072.689,-19.874,438.821,172.967,22.869,154.095
C08617=1072.696,-19.625,438.807,172.969,22.872,154.095
C08618=1072.702,-19.376,438.794,172.970,22.874,154.096
C08619=1072.707,-19.125,438.781,172.971,22.876,154.096
C08620=1072.713,-18.876,438.768,172.973,22.879,154.096
C08621=1072.720,-18.627,438.755,172.975,22.882,154.096
C08622=1072.725,-18.377,438.741,172.976,22.884,154.097
C08623=1072.731,-18.128,438.727,172.977,22.886,154.097
C08624=1072.738,-17.851,438.712,172.979,22.888,154.097
C08625=1072.744,-17.574,438.697,172.981,22.891,154.097
C08626=1072.752,-17.297,438.683,172.982,22.894,154.098
C08627=1072.758,-17.021,438.668,172.983,22.896,154.098
C08628=1072.764,-16.771,438.655,172.985,22.898,154.098
C08629=1072.770,-16.521,438.642,172.986,22.901,154.098
C08630=1072.776,-16.271,438.628,172.988,22.903,154.099
C08631=1072.782,-16.022,438.614,172.989,22.906,154.099
C08632=1072.788,-15.773,438.601,172.991,22.908,154.099
C08633=1072.794,-15.523,438.588,172.992,22.910,154.099
C08634=1072.800,-15.274,438.574,172.993,22.912,154.100
C08635=1072.806,-15.024,438.560,172.995,22.915,154.100
C08636=1072.813,-14.775,438.547,172.996,22.917,154.100
C08637=1072.818,-14.524,438.534,172.997,22.920,154.100
C08638=1072.824,-14.275,438.520,172.998,22.922,154.101
C08639=1072.830,-14.025,438.506,173.001,22.924,154.101
C08640=1072.836,-13.776,438.493,173.002,22.927,154.101
C08641=1072.841,-13.527,438.479,173.003,22.929,154.101
C08642=1072.847,-13.277,438.465,173.005,22.932,154.102
C08643=1072.854,-13.027,438.452,173.006,22.934,154.102
C08644=1072.859,-12.778,438.438,173.007,22.937,154.102
C08645=1072.865,-12.528,438.425,173.009,22.938,154.102
C08646=1072.871,-12.279,438.411,173.010,22.941,154.103
C08647=1072.877,-12.029,438.398,173.011,22.943,154.103
C08648=1072.882,-11.780,438.384,173.013,22.946,154.103
C08649=1072.889,-11.530,438.370,173.014,22.949,154.103
C08650=1072.895,-11.280,438.356,173.016,22.951,154.104
C08651=1072.901,-11.031,438.343,173.017,22.954,154.104
C08652=1072.906,-10.781,438.329,173.018,22.955,154.104
C08653=1072.912,-10.532,438.315,173.020,22.958,154.104
C08654=1072.919,-10.282,438.302,173.021,22.960,154.105
C08655=1072.924,-10.032,438.288,173.022,22.963,154.105
C08656=1072.930,-9.783,438.274,173.024,22.965,154.105
C08657=1072.936,-9.534,438.261,173.026,22.968,154.106
C08658=1072.943,-9.284,438.246,173.027,22.970,154.106
C08659=1072.948,-9.035,438.232,173.028,22.972,154.106
C08660=1072.954,-8.785,438.219,173.030,22.975,154.106
C08661=1072.960,-8.536,438.205,173.031,22.977,154.107
C08662=1072.966,-8.286,438.191,173.032,22.980,154.107
C08663=1072.972,-8.036,438.178,173.033,22.982,154.107
C08664=1072.978,-7.787,438.164,173.035,22.984,154.107
C08665=1072.983,-7.537,438.150,173.036,22.987,154.108
C08666=1072.990,-7.287,438.136,173.038,22.989,154.108
C08667=1072.996,-7.038,438.122,173.040,22.992,154.108
C08668=1073.002,-6.789,438.109,173.041,22.994,154.108
C08669=1073.008,-6.539,438.095,173.042,22.996,154.109
C08670=1073.014,-6.289,438.080,173.043,22.999,154.109
C08671=1073.020,-6.040,438.067,173.045,23.001,154.109
C08672=1073.025,-5.790,438.053,173.046,23.004,154.109
C08673=1073.032,-5.542,438.039,173.047,23.006,154.110
C08674=1073.038,-5.291,438.025,173.050,23.008,154.110
C08675=1073.044,-5.042,438.011,173.051,23.011,154.110
C08676=1073.050,-4.792,437.998,173.052,23.013,154.110
C08677=1073.056,-4.542,437.984,173.053,23.016,154.111
C08678=1073.062,-4.293,437.969,173.055,23.018,154.111
C08679=1073.068,-4.044,437.956,173.056,23.021,154.111
C08680=1073.074,-3.794,437.942,173.057,23.023,154.111
C08681=1073.080,-3.544,437.928,173.059,23.025,154.112
C08682=1073.086,-3.295,437.914,173.060,23.027,154.112
C08683=1073.092,-3.045,437.900,173.062,23.030,154.112
C08684=1073.097,-2.796,437.886,173.063,23.033,154.113
C08685=1073.103,-2.547,437.871,173.065,23.035,154.113
C08686=1073.109,-2.297,437.857,173.066,23.037,154.113
C08687=1073.116,-2.047,437.844,173.067,23.040,154.113
C08688=1073.121,-1.769,437.828,173.068,23.043,154.114
C08689=1073.128,-1.491,437.812,173.070,23.046,154.114
C08690=1073.134,-1.212,437.796,173.072,23.048,154.114
C08691=1073.141,-0.934,437.780,173.073,23.051,154.115
C08692=1073.147,-0.685,437.766,173.075,23.054,154.115
C08693=1073.153,-0.434,437.752,173.076,23.056,154.115
C08694=1073.159,-0.185,437.737,173.078,23.059,154.116
C08695=1073.164,0.064,437.724,173.079,23.061,154.116
C08696=1073.170,0.314,437.710,173.080,23.064,154.116
C08697=1073.176,0.564,437.695,173.081,23.066,154.116
C08698=1073.182,0.813,437.682,173.083,23.069,154.117
C08699=1073.188,1.062,437.668,173.084,23.071,154.117
C08700=1073.194,1.312,437.653,173.086,23.074,154.117
C08701=1073.200,1.562,437.639,173.087,23.076,154.117
C08702=1073.205,1.811,437.624,173.089,23.079,154.118
C08703=1073.212,2.061,437.610,173.090,23.081,154.118
C08704=1073.217,2.310,437.595,173.091,23.083,154.118
C08705=1073.223,2.559,437.582,173.092,23.086,154.119
C08706=1073.229,2.810,437.567,173.094,23.088,154.119
C08707=1073.235,3.059,437.553,173.095,23.091,154.119
C08708=1073.241,3.309,437.539,173.097,23.094,154.119
C08709=1073.247,3.558,437.524,173.098,23.096,154.120
C08710=1073.252,3.807,437.510,173.100,23.098,154.120
C08711=1073.259,4.057,437.496,173.101,23.101,154.120
C08712=1073.265,4.306,437.482,173.102,23.103,154.121
C08713=1073.270,4.555,437.467,173.104,23.106,154.121
C08714=1073.276,4.806,437.453,173.105,23.108,154.121
C08715=1073.282,5.055,437.439,173.106,23.111,154.121
C08716=1073.288,5.305,437.424,173.107,23.113,154.122
C08717=1073.294,5.554,437.410,173.110,23.116,154.122
C08718=1073.300,5.804,437.395,173.111,23.118,154.122
C08719=1073.306,6.053,437.381,173.112,23.121,154.123
C08720=1073.312,6.302,437.366,173.113,23.123,154.123
C08721=1073.318,6.552,437.352,173.115,23.126,154.123
C08722=1073.324,6.801,437.337,173.116,23.128,154.123
C08723=1073.330,7.051,437.323,173.117,23.130,154.124
C08724=1073.335,7.300,437.309,173.118,23.133,154.124
C08725=1073.342,7.551,437.294,173.121,23.136,154.124
C08726=1073.347,7.800,437.280,173.122,23.138,154.124
C08727=1073.353,8.049,437.265,173.123,23.141,154.125
C08728=1073.359,8.299,437.251,173.124,23.143,154.125
C08729=1073.365,8.548,437.236,173.126,23.146,154.125
C08730=1073.371,8.798,437.222,173.127,23.148,154.126
C08731=1073.377,9.047,437.208,173.128,23.151,154.126
C08732=1073.383,9.297,437.193,173.129,23.153,154.126
C08733=1073.389,9.546,437.179,173.132,23.156,154.127
C08734=1073.395,9.796,437.164,173.133,23.158,154.127
C08735=1073.401,10.045,437.149,173.134,23.161,154.127
C08736=1073.407,10.295,437.135,173.135,23.163,154.127
C08737=1073.413,10.544,437.121,173.137,23.166,154.128
C08738=1073.419,10.794,437.106,173.138,23.168,154.128
C08739=1073.425,11.043,437.091,173.139,23.170,154.128
C08740=1073.431,11.293,437.077,173.141,23.173,154.129
C08741=1073.437,11.542,437.062,173.143,23.176,154.129
C08742=1073.443,11.792,437.047,173.144,23.178,154.129
C08743=1073.449,12.041,437.033,173.145,23.181,154.129
C08744=1073.455,12.291,437.018,173.147,23.183,154.130
C08745=1073.461,12.540,437.004,173.148,23.185,154.130
C08746=1073.467,12.789,436.989,173.149,23.188,154.130
C08747=1073.473,13.040,436.975,173.150,23.190,154.130
C08748=1073.479,13.289,436.960,173.152,23.193,154.131
C08749=1073.485,13.538,436.945,173.154,23.195,154.131
C08750=1073.491,13.787,436.931,173.155,23.198,154.131
C08751=1073.498,14.037,436.916,173.156,23.200,154.132
C08752=1073.503,14.317,436.899,173.158,23.203,154.132
C08753=1073.511,14.598,436.882,173.160,23.206,154.132
C08754=1073.517,14.878,436.865,173.161,23.208,154.133
C08755=1073.524,15.158,436.849,173.162,23.211,154.133
C08756=1073.530,15.408,436.835,173.164,23.214,154.133
C08757=1073.535,15.658,436.820,173.166,23.217,154.133
C08758=1073.541,15.907,436.805,173.167,23.219,154.134
C08759=1073.547,16.156,436.790,173.168,23.222,154.134
C08760=1073.553,16.406,436.775,173.169,23.224,154.134
C08761=1073.559,16.655,436.760,173.171,23.227,154.135
C08762=1073.565,16.905,436.745,173.172,23.229,154.135
C08763=1073.570,17.154,436.731,173.173,23.232,154.135
C08764=1073.577,17.404,436.717,173.175,23.235,154.136
C08765=1073.582,17.654,436.701,173.177,23.237,154.136
C08766=1073.588,17.903,436.686,173.178,23.239,154.136
C08767=1073.595,18.153,436.671,173.179,23.242,154.136
C08768=1073.600,18.402,436.656,173.180,23.244,154.137
C08769=1073.606,18.652,436.641,173.182,23.247,154.137
C08770=1073.612,18.901,436.627,173.183,23.250,154.137
C08771=1073.618,19.150,436.612,173.185,23.252,154.138
C08772=1073.624,19.400,436.596,173.186,23.255,154.138
C08773=1073.630,19.649,436.582,173.188,23.257,154.138
C08774=1073.636,19.899,436.567,173.189,23.260,154.138
C08775=1073.642,20.148,436.552,173.190,23.262,154.139
C08776=1073.647,20.398,436.537,173.191,23.265,154.139
C08777=1073.654,20.647,436.522,173.193,23.267,154.139
C08778=1073.659,20.897,436.507,173.194,23.270,154.140
C08779=1073.665,21.146,436.492,173.196,23.273,154.140
C08780=1073.671,21.395,436.477,173.197,23.275,154.140
C08781=1073.677,21.645,436.461,173.199,23.278,154.141
C08782=1073.683,21.895,436.447,173.200,23.280,154.141
C08783=1073.688,22.144,436.431,173.201,23.282,154.141
C08784=1073.694,22.394,436.416,173.202,23.285,154.142
C08785=1073.701,22.643,436.401,173.204,23.288,154.142
C08786=1073.706,22.893,436.386,173.206,23.291,154.142
C08787=1073.712,23.142,436.371,173.207,23.293,154.142
C08788=1073.717,23.392,436.356,173.208,23.295,154.143
C08789=1073.724,23.641,436.341,173.210,23.298,154.143
C08790=1073.730,23.891,436.326,173.211,23.301,154.143
C08791=1073.735,24.140,436.310,173.212,23.303,154.144
C08792=1073.742,24.389,436.295,173.213,23.306,154.144
C08793=1073.747,24.639,436.280,173.215,23.308,154.144
C08794=1073.753,24.888,436.265,173.217,23.311,154.144
C08795=1073.759,25.138,436.250,173.218,23.313,154.145
C08796=1073.765,25.388,436.235,173.219,23.316,154.145
C08797=1073.771,25.637,436.220,173.221,23.319,154.145
C08798=1073.777,25.886,436.204,173.222,23.321,154.146
C08799=1073.783,26.136,436.189,173.223,23.323,154.146
C08800=1073.788,26.385,436.174,173.224,23.326,154.146
C08801=1073.795,26.635,436.159,173.227,23.329,154.147
C08802=1073.800,26.885,436.143,173.228,23.331,154.147
C08803=1073.807,27.133,436.128,173.229,23.333,154.147
C08804=1073.812,27.383,436.113,173.230,23.336,154.148
C08805=1073.819,27.633,436.098,173.232,23.339,154.148
C08806=1073.824,27.883,436.082,173.233,23.341,154.148
C08807=1073.830,28.132,436.067,173.234,23.344,154.148
C08808=1073.836,28.381,436.051,173.236,23.346,154.149
C08809=1073.842,28.631,436.036,173.238,23.349,154.149
C08810=1073.847,28.880,436.021,173.239,23.352,154.149
C08811=1073.854,29.129,436.006,173.240,23.354,154.150
C08812=1073.860,29.379,435.990,173.241,23.357,154.150
C08813=1073.865,29.628,435.975,173.243,23.359,154.150
C08814=1073.871,29.878,435.960,173.244,23.361,154.150
C08815=1073.877,30.127,435.944,173.246,23.365,154.151
C08816=1073.884,30.409,435.927,173.247,23.367,154.151
C08817=1073.890,30.691,435.909,173.248,23.370,154.152
C08818=1073.897,30.972,435.892,173.250,23.373,154.152
C08819=1073.903,31.254,435.874,173.252,23.376,154.152
C08820=1073.909,31.503,435.859,173.253,23.378,154.152
C08821=1073.915,31.753,435.843,173.255,23.382,154.153
C08822=1073.920,32.002,435.827,173.256,23.384,154.153
C08823=1073.927,32.252,435.812,173.258,23.386,154.153
C08824=1073.932,32.502,435.797,173.259,23.389,154.154
C08825=1073.938,32.751,435.781,173.260,23.391,154.154
C08826=1073.944,33.000,435.766,173.261,23.394,154.154
C08827=1073.950,33.250,435.750,173.263,23.397,154.155
C08828=1073.956,33.499,435.734,173.265,23.399,154.155
C08829=1073.962,33.749,435.719,173.266,23.402,154.155
C08830=1073.968,33.997,435.703,173.268,23.404,154.156
C08831=1073.973,34.247,435.688,173.269,23.407,154.156
C08832=1073.980,34.496,435.672,173.270,23.410,154.156
C08833=1073.986,34.746,435.657,173.271,23.412,154.157
C08834=1073.991,34.996,435.641,173.273,23.415,154.157
C08835=1073.997,35.245,435.626,173.275,23.417,154.157
C08836=1074.003,35.495,435.610,173.276,23.420,154.157
C08837=1074.009,35.744,435.594,173.277,23.423,154.158
C08838=1074.015,35.994,435.579,173.278,23.425,154.158
C08839=1074.021,36.243,435.563,173.280,23.427,154.158
C08840=1074.026,36.492,435.548,173.281,23.430,154.159
C08841=1074.033,36.741,435.532,173.283,23.433,154.159
C08842=1074.039,36.991,435.516,173.284,23.436,154.159
C08843=1074.045,37.241,435.500,173.286,23.438,154.160
C08844=1074.050,37.491,435.485,173.287,23.440,154.160
C08845=1074.057,37.740,435.469,173.288,23.443,154.160
C08846=1074.062,37.988,435.453,173.290,23.445,154.160
C08847=1074.068,38.238,435.438,173.292,23.448,154.161
C08848=1074.074,38.488,435.421,173.293,23.451,154.161
C08849=1074.079,38.738,435.406,173.294,23.453,154.161
C08850=1074.085,38.987,435.390,173.296,23.456,154.162
C08851=1074.091,39.236,435.375,173.297,23.459,154.162
C08852=1074.097,39.485,435.359,173.298,23.461,154.162
C08853=1074.103,39.735,435.342,173.300,23.464,154.163
C08854=1074.109,39.985,435.327,173.301,23.466,154.163
C08855=1074.115,40.234,435.311,173.303,23.469,154.163
C08856=1074.120,40.484,435.295,173.304,23.472,154.164
C08857=1074.126,40.733,435.279,173.305,23.474,154.164
C08858=1074.132,40.982,435.263,173.307,23.476,154.164
C08859=1074.137,41.232,435.247,173.308,23.479,154.165
C08860=1074.144,41.481,435.232,173.310,23.482,154.165
C08861=1074.150,41.730,435.215,173.311,23.485,154.165
C08862=1074.156,41.980,435.200,173.312,23.487,154.165
C08863=1074.161,42.230,435.184,173.314,23.489,154.166
C08864=1074.167,42.478,435.168,173.315,23.492,154.166
C08865=1074.172,42.728,435.152,173.316,23.495,154.166
C08866=1074.178,42.978,435.136,173.318,23.497,154.167
C08867=1074.184,43.227,435.120,173.320,23.500,154.167
C08868=1074.190,43.476,435.103,173.321,23.503,154.167
C08869=1074.196,43.726,435.088,173.322,23.505,154.168
C08870=1074.202,43.976,435.072,173.323,23.508,154.168
C08871=1074.208,44.225,435.055,173.325,23.510,154.168
C08872=1074.213,44.474,435.040,173.327,23.513,154.169
C08873=1074.219,44.724,435.024,173.328,23.516,154.169
C08874=1074.225,44.973,435.008,173.329,23.518,154.169
C08875=1074.231,45.222,434.991,173.331,23.521,154.170
C08876=1074.237,45.472,434.975,173.332,23.524,154.170
C08877=1074.242,45.722,434.960,173.333,23.526,154.170
C08878=1074.247,45.971,434.943,173.335,23.529,154.170
C08879=1074.253,46.220,434.927,173.337,23.532,154.171
C08880=1074.259,46.502,434.909,173.338,23.535,154.171
C08881=1074.267,46.784,434.890,173.340,23.537,154.171
C08882=1074.273,47.065,434.872,173.341,23.540,154.172
C08883=1074.279,47.347,434.854,173.343,23.544,154.172
C08884=1074.285,47.597,434.838,173.344,23.546,154.173
C08885=1074.291,47.846,434.821,173.346,23.548,154.173
C08886=1074.297,48.095,434.805,173.347,23.551,154.173
C08887=1074.302,48.344,434.789,173.348,23.554,154.174
C08888=1074.308,48.594,434.772,173.350,23.557,154.174
C08889=1074.313,48.844,434.757,173.351,23.559,154.174
C08890=1074.319,49.093,434.740,173.353,23.562,154.174
C08891=1074.325,49.342,434.724,173.354,23.564,154.175
C08892=1074.331,49.592,434.708,173.355,23.567,154.175
C08893=1074.337,49.841,434.692,173.357,23.570,154.175
C08894=1074.342,50.091,434.675,173.359,23.572,154.176
C08895=1074.348,50.340,434.659,173.360,23.575,154.176
C08896=1074.354,50.589,434.642,173.361,23.578,154.176
C08897=1074.360,50.839,434.626,173.363,23.580,154.177
C08898=1074.366,51.088,434.610,173.364,23.583,154.177
C08899=1074.372,51.337,434.594,173.365,23.585,154.177
C08900=1074.377,51.587,434.577,173.367,23.588,154.178
C08901=1074.383,51.836,434.560,173.368,23.591,154.178
C08902=1074.389,52.086,434.544,173.370,23.593,154.178
C08903=1074.395,52.335,434.528,173.371,23.595,154.179
C08904=1074.401,52.584,434.512,173.372,23.598,154.179
C08905=1074.406,52.834,434.495,173.374,23.601,154.179
C08906=1074.412,53.083,434.479,173.376,23.604,154.179
C08907=1074.418,53.333,434.462,173.377,23.606,154.180
C08908=1074.424,53.582,434.446,173.378,23.609,154.180
C08909=1074.430,53.831,434.430,173.380,23.611,154.180
C08910=1074.435,54.081,434.413,173.381,23.614,154.181
C08911=1074.441,54.330,434.397,173.383,23.616,154.181
C08912=1074.447,54.580,434.380,173.384,23.619,154.181
C08913=1074.453,54.829,434.364,173.386,23.622,154.182
C08914=1074.459,55.079,434.348,173.387,23.624,154.182
C08915=1074.465,55.328,434.330,173.388,23.627,154.182
C08916=1074.471,55.577,434.314,173.390,23.629,154.183
C08917=1074.477,55.826,434.298,173.392,23.632,154.183
C08918=1074.483,56.076,434.282,173.393,23.635,154.183
C08919=1074.488,56.325,434.265,173.394,23.637,154.183
C08920=1074.494,56.575,434.249,173.395,23.639,154.184
C08921=1074.500,56.824,434.232,173.398,23.643,154.184
C08922=1074.506,57.073,434.215,173.399,23.645,154.184
C08923=1074.511,57.322,434.198,173.400,23.648,154.185
C08924=1074.517,57.572,434.182,173.401,23.650,154.185
C08925=1074.524,57.822,434.166,173.403,23.652,154.185
C08926=1074.530,58.071,434.149,173.404,23.655,154.186
C08927=1074.535,58.321,434.132,173.406,23.658,154.186
C08928=1074.541,58.569,434.115,173.407,23.660,154.186
C08929=1074.547,58.819,434.099,173.409,23.663,154.187
C08930=1074.553,59.068,434.083,173.410,23.665,154.187
C08931=1074.558,59.318,434.066,173.411,23.668,154.187
C08932=1074.564,59.567,434.049,173.413,23.671,154.188
C08933=1074.570,59.816,434.033,173.415,23.673,154.188
C08934=1074.576,60.066,434.016,173.416,23.676,154.188
C08935=1074.582,60.316,433.999,173.417,23.678,154.188
C08936=1074.588,60.564,433.982,173.419,23.680,154.189
C08937=1074.594,60.814,433.966,173.421,23.683,154.189
C08938=1074.600,61.063,433.949,173.422,23.686,154.189
C08939=1074.605,61.313,433.933,173.423,23.689,154.190
C08940=1074.612,61.562,433.916,173.425,23.691,154.190
C08941=1074.618,61.812,433.899,173.426,23.693,154.190
C08942=1074.624,62.061,433.883,173.428,23.696,154.190
C08943=1074.630,62.310,433.866,173.430,23.699,154.191
C08944=1074.636,62.591,433.847,173.431,23.701,154.191
C08945=1074.643,62.873,433.827,173.433,23.704,154.191
C08946=1074.650,63.154,433.809,173.434,23.707,154.192
C08947=1074.656,63.436,433.790,173.436,23.710,154.192
C08948=1074.662,63.685,433.774,173.438,23.713,154.192
C08949=1074.668,63.935,433.756,173.439,23.715,154.193
C08950=1074.674,64.184,433.739,173.440,23.718,154.193
C08951=1074.680,64.433,433.723,173.442,23.720,154.193
C08952=1074.686,64.683,433.706,173.444,23.723,154.194
C08953=1074.692,64.932,433.689,173.445,23.726,154.194
C08954=1074.698,65.182,433.672,173.446,23.728,154.194
C08955=1074.704,65.431,433.655,173.448,23.730,154.195
C08956=1074.709,65.681,433.638,173.450,23.733,154.195
C08957=1074.715,65.929,433.621,173.451,23.736,154.195
C08958=1074.720,66.179,433.604,173.452,23.739,154.196
C08959=1074.727,66.428,433.587,173.454,23.741,154.196
C08960=1074.733,66.678,433.570,173.456,23.744,154.196
C08961=1074.738,66.927,433.553,173.457,23.746,154.196
C08962=1074.744,67.176,433.536,173.458,23.749,154.197
C08963=1074.750,67.426,433.519,173.460,23.751,154.197
C08964=1074.755,67.675,433.503,173.461,23.754,154.197
C08965=1074.762,67.925,433.485,173.463,23.757,154.198
C08966=1074.768,68.174,433.468,173.464,23.759,154.198
C08967=1074.773,68.423,433.451,173.466,23.762,154.198
C08968=1074.778,68.673,433.434,173.467,23.764,154.199
C08969=1074.785,68.921,433.417,173.468,23.767,154.199
C08970=1074.790,69.172,433.400,173.471,23.769,154.199
C08971=1074.797,69.420,433.383,173.472,23.772,154.199
C08972=1074.802,69.670,433.366,173.473,23.775,154.200
C08973=1074.807,69.919,433.348,173.474,23.777,154.200
C08974=1074.814,70.169,433.331,173.477,23.780,154.200
C08975=1074.819,70.418,433.314,173.478,23.782,154.201
C08976=1074.825,70.667,433.297,173.479,23.785,154.201
C08977=1074.831,70.917,433.280,173.480,23.788,154.201
C08978=1074.836,71.166,433.263,173.482,23.790,154.202
C08979=1074.843,71.415,433.245,173.484,23.793,154.202
C08980=1074.848,71.665,433.229,173.485,23.795,154.202
C08981=1074.854,71.914,433.211,173.486,23.798,154.203
C08982=1074.860,72.163,433.193,173.488,23.800,154.203
C08983=1074.865,72.413,433.176,173.490,23.803,154.203
C08984=1074.872,72.662,433.159,173.491,23.805,154.203
C08985=1074.877,72.911,433.142,173.492,23.808,154.204
C08986=1074.882,73.161,433.125,173.494,23.811,154.204
C08987=1074.888,73.410,433.107,173.495,23.813,154.204
C08988=1074.895,73.659,433.090,173.497,23.816,154.205
C08989=1074.900,73.909,433.073,173.499,23.818,154.205
C08990=1074.906,74.159,433.055,173.500,23.821,154.205
C08991=1074.912,74.408,433.038,173.501,23.824,154.206
C08992=1074.918,74.656,433.021,173.503,23.826,154.206
C08993=1074.923,74.906,433.004,173.505,23.829,154.206
C08994=1074.929,75.156,432.986,173.506,23.831,154.207
C08995=1074.935,75.405,432.968,173.507,23.834,154.207
C08996=1074.941,75.653,432.951,173.509,23.837,154.207
C08997=1074.947,75.904,432.934,173.511,23.839,154.207
C08998=1074.952,76.153,432.917,173.512,23.842,154.208
C08999=1074.958,76.402,432.899,173.513,23.844,154.208
C09000=1074.964,76.652,432.881,173.515,23.847,154.208
C09001=1074.970,76.900,432.864,173.517,23.850,154.209
C09002=1074.976,77.149,432.847,173.518,23.852,154.209
C09003=1074.981,77.400,432.829,173.520,23.854,154.209
C09004=1074.987,77.649,432.812,173.521,23.857,154.210
C09005=1074.993,77.898,432.794,173.523,23.860,154.210
C09006=1074.999,78.147,432.777,173.524,23.862,154.210
C09007=1075.005,78.396,432.759,173.526,23.865,154.211
C09008=1075.011,78.678,432.740,173.528,23.868,154.211
C09009=1075.018,78.959,432.720,173.529,23.870,154.211
C09010=1075.024,79.240,432.699,173.531,23.874,154.212
C09011=1075.030,79.523,432.680,173.532,23.876,154.212
C09012=1075.036,79.772,432.662,173.534,23.879,154.212
C09013=1075.041,80.021,432.645,173.536,23.882,154.213
C09014=1075.048,80.270,432.627,173.537,23.884,154.213
C09015=1075.053,80.519,432.609,173.538,23.887,154.213
C09016=1075.059,80.768,432.592,173.541,23.890,154.213
C09017=1075.065,81.018,432.574,173.542,23.892,154.214
C09018=1075.070,81.267,432.556,173.543,23.895,154.214
C09019=1075.076,81.516,432.539,173.545,23.897,154.214
C09020=1075.082,81.766,432.521,173.547,23.900,154.215
C09021=1075.087,82.015,432.503,173.548,23.903,154.215
C09022=1075.093,82.264,432.485,173.549,23.905,154.215
C09023=1075.099,82.514,432.468,173.551,23.907,154.216
C09024=1075.105,82.763,432.450,173.553,23.910,154.216
C09025=1075.111,83.013,432.432,173.554,23.913,154.216
C09026=1075.116,83.262,432.414,173.555,23.915,154.217
C09027=1075.122,83.511,432.397,173.557,23.918,154.217
C09028=1075.128,83.760,432.379,173.559,23.921,154.217
C09029=1075.133,84.009,432.361,173.560,23.923,154.217
C09030=1075.139,84.259,432.343,173.562,23.925,154.218
C09031=1075.145,84.508,432.326,173.563,23.928,154.218
C09032=1075.150,84.757,432.308,173.565,23.931,154.218
C09033=1075.157,85.007,432.290,173.566,23.933,154.219
C09034=1075.162,85.256,432.273,173.568,23.936,154.219
C09035=1075.168,85.506,432.255,173.569,23.938,154.219
C09036=1075.174,85.755,432.237,173.571,23.941,154.219
C09037=1075.180,86.003,432.219,173.572,23.944,154.220
C09038=1075.186,86.253,432.201,173.574,23.946,154.220
C09039=1075.190,86.502,432.183,173.575,23.949,154.220
C09040=1075.197,86.752,432.165,173.577,23.951,154.221
C09041=1075.202,87.001,432.147,173.579,23.954,154.221
C09042=1075.208,87.251,432.130,173.580,23.956,154.221
C09043=1075.214,87.500,432.112,173.582,23.959,154.222
C09044=1075.220,87.749,432.093,173.583,23.962,154.222
C09045=1075.226,87.998,432.076,173.585,23.964,154.222
C09046=1075.232,88.248,432.058,173.586,23.966,154.223
C09047=1075.237,88.497,432.040,173.588,23.969,154.223
C09048=1075.243,88.747,432.022,173.590,23.972,154.223
C09049=1075.249,88.995,432.004,173.591,23.974,154.223
C09050=1075.255,89.245,431.986,173.592,23.976,154.224
C09051=1075.260,89.494,431.968,173.595,23.979,154.224
C09052=1075.266,89.744,431.950,173.596,23.981,154.224
C09053=1075.272,89.992,431.932,173.597,23.984,154.225
C09054=1075.278,90.242,431.914,173.599,23.987,154.225
C09055=1075.284,90.491,431.896,173.601,23.989,154.225
C09056=1075.290,90.741,431.878,173.602,23.992,154.225
C09057=1075.296,90.989,431.860,173.603,23.994,154.226
C09058=1075.301,91.239,431.841,173.606,23.997,154.226
C09059=1075.307,91.488,431.824,173.607,23.999,154.226
C09060=1075.313,91.737,431.805,173.608,24.002,154.227
C09061=1075.318,91.987,431.787,173.610,24.005,154.227
C09062=1075.324,92.237,431.769,173.612,24.007,154.227
C09063=1075.330,92.485,431.751,173.613,24.010,154.228
C09064=1075.335,92.735,431.732,173.615,24.012,154.228
C09065=1075.341,92.984,431.715,173.617,24.015,154.228
C09066=1075.347,93.233,431.696,173.618,24.018,154.229
C09067=1075.352,93.483,431.678,173.619,24.020,154.229
C09068=1075.358,93.732,431.660,173.622,24.023,154.229
C09069=1075.364,93.981,431.642,173.623,24.025,154.229
C09070=1075.369,94.231,431.623,173.624,24.027,154.230
C09071=1075.375,94.479,431.605,173.626,24.030,154.230
C09072=1075.382,94.761,431.585,173.628,24.033,154.230
C09073=1075.388,95.043,431.564,173.630,24.036,154.231
C09074=1075.395,95.324,431.543,173.631,24.039,154.231
C09075=1075.401,95.605,431.523,173.633,24.042,154.231
C09076=1075.407,95.855,431.504,173.635,24.044,154.232
C09077=1075.412,96.104,431.486,173.636,24.047,154.232
C09078=1075.419,96.353,431.468,173.638,24.050,154.232
C09079=1075.424,96.603,431.449,173.639,24.052,154.232
C09080=1075.430,96.851,431.431,173.641,24.054,154.233
C09081=1075.436,97.101,431.413,173.643,24.057,154.233
C09082=1075.441,97.350,431.394,173.644,24.059,154.233
C09083=1075.447,97.599,431.376,173.646,24.062,154.234
C09084=1075.453,97.849,431.357,173.647,24.065,154.234
C09085=1075.458,98.098,431.339,173.649,24.067,154.234
C09086=1075.465,98.347,431.321,173.651,24.070,154.235
C09087=1075.470,98.596,431.302,173.652,24.072,154.235
C09088=1075.476,98.845,431.284,173.654,24.075,154.235
C09089=1075.482,99.095,431.265,173.656,24.077,154.235
C09090=1075.487,99.344,431.247,173.657,24.080,154.236
C09091=1075.494,99.593,431.228,173.659,24.082,154.236
C09092=1075.499,99.843,431.210,173.660,24.085,154.236
C09093=1075.505,100.092,431.192,173.662,24.087,154.237
C09094=1075.510,100.342,431.173,173.664,24.090,154.237
C09095=1075.517,100.591,431.154,173.665,24.092,154.237
C09096=1075.522,100.839,431.136,173.667,24.094,154.237
C09097=1075.528,101.089,431.118,173.668,24.097,154.238
C09098=1075.534,101.338,431.099,173.670,24.100,154.238
C09099=1075.539,101.587,431.080,173.672,24.102,154.238
C09100=1075.545,101.837,431.062,173.673,24.105,154.239
C09101=1075.551,102.086,431.043,173.675,24.108,154.239
C09102=1075.556,102.335,431.024,173.677,24.110,154.239
C09103=1075.562,102.585,431.006,173.678,24.112,154.239
C09104=1075.567,102.833,430.987,173.680,24.115,154.240
C09105=1075.573,103.083,430.968,173.681,24.118,154.240
C09106=1075.580,103.332,430.949,173.683,24.120,154.240
